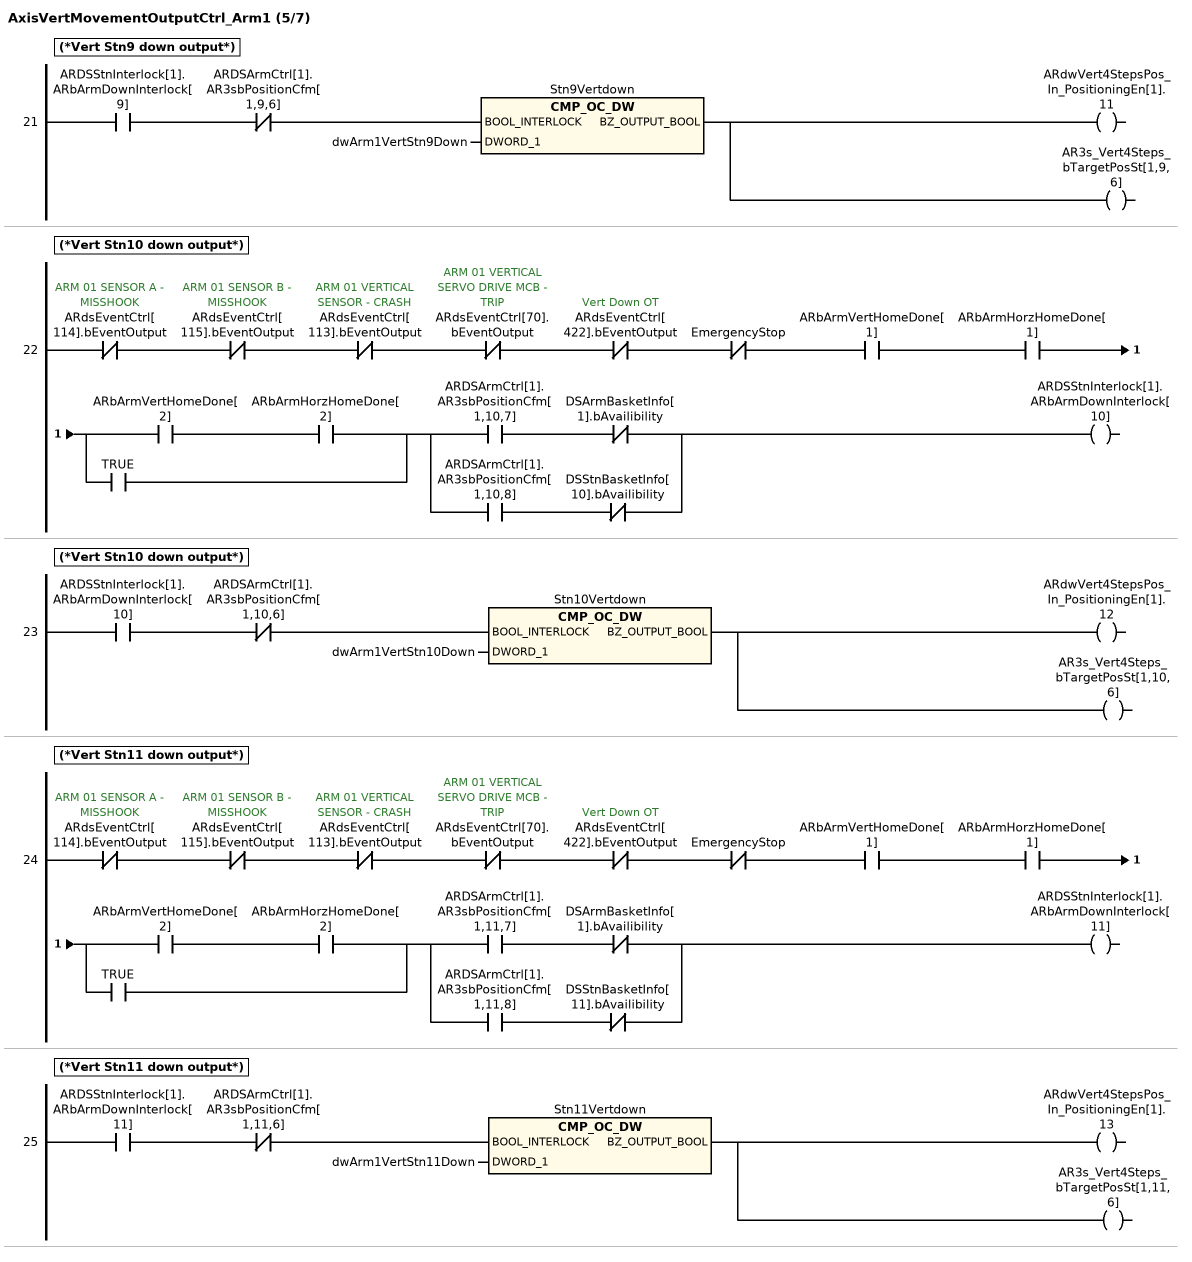
// NETWORK 21
// label: (*Vert Stn9 down output*)
Stn9Vertdown(BOOL_INTERLOCK := ARDSStnInterlock[1].ARbArmDownInterlock[9] AND NOT ARDSArmCtrl[1].AR3sbPositionCfm[1,9,6], DWORD_1 := dwArm1VertStn9Down); // CMP_OC_DW
ARdwVert4StepsPos_In_PositioningEn[1].11 := Stn9Vertdown.BZ_OUTPUT_BOOL;
AR3s_Vert4Steps_bTargetPosSt[1,9,6] := Stn9Vertdown.BZ_OUTPUT_BOOL;

// NETWORK 22
//   ARdsEventCtrl[114].bEventOutput: ARM 01 SENSOR A - MISSHOOK
//   ARdsEventCtrl[115].bEventOutput: ARM 01 SENSOR B - MISSHOOK
//   ARdsEventCtrl[113].bEventOutput: ARM 01 VERTICAL SENSOR - CRASH
//   ARdsEventCtrl[70].bEventOutput: ARM 01 VERTICAL SERVO DRIVE MCB - TRIP
//   ARdsEventCtrl[422].bEventOutput: Vert Down OT
// label: (*Vert Stn10 down output*)
ARDSStnInterlock[1].ARbArmDownInterlock[10] := (NOT ARdsEventCtrl[114].bEventOutput AND NOT ARdsEventCtrl[115].bEventOutput AND NOT ARdsEventCtrl[113].bEventOutput AND NOT ARdsEventCtrl[70].bEventOutput AND NOT ARdsEventCtrl[422].bEventOutput AND NOT EmergencyStop) AND ARbArmVertHomeDone[1] AND ARbArmHorzHomeDone[1] AND (ARbArmVertHomeDone[2] AND ARbArmHorzHomeDone[2] OR TRUE) AND (ARDSArmCtrl[1].AR3sbPositionCfm[1,10,7] AND NOT DSArmBasketInfo[1].bAvailibility OR ARDSArmCtrl[1].AR3sbPositionCfm[1,10,8] AND NOT DSStnBasketInfo[10].bAvailibility);

// NETWORK 23
// label: (*Vert Stn10 down output*)
Stn10Vertdown(BOOL_INTERLOCK := ARDSStnInterlock[1].ARbArmDownInterlock[10] AND NOT ARDSArmCtrl[1].AR3sbPositionCfm[1,10,6], DWORD_1 := dwArm1VertStn10Down); // CMP_OC_DW
ARdwVert4StepsPos_In_PositioningEn[1].12 := Stn10Vertdown.BZ_OUTPUT_BOOL;
AR3s_Vert4Steps_bTargetPosSt[1,10,6] := Stn10Vertdown.BZ_OUTPUT_BOOL;

// NETWORK 24
//   ARdsEventCtrl[114].bEventOutput: ARM 01 SENSOR A - MISSHOOK
//   ARdsEventCtrl[115].bEventOutput: ARM 01 SENSOR B - MISSHOOK
//   ARdsEventCtrl[113].bEventOutput: ARM 01 VERTICAL SENSOR - CRASH
//   ARdsEventCtrl[70].bEventOutput: ARM 01 VERTICAL SERVO DRIVE MCB - TRIP
//   ARdsEventCtrl[422].bEventOutput: Vert Down OT
// label: (*Vert Stn11 down output*)
ARDSStnInterlock[1].ARbArmDownInterlock[11] := (NOT ARdsEventCtrl[114].bEventOutput AND NOT ARdsEventCtrl[115].bEventOutput AND NOT ARdsEventCtrl[113].bEventOutput AND NOT ARdsEventCtrl[70].bEventOutput AND NOT ARdsEventCtrl[422].bEventOutput AND NOT EmergencyStop) AND ARbArmVertHomeDone[1] AND ARbArmHorzHomeDone[1] AND (ARbArmVertHomeDone[2] AND ARbArmHorzHomeDone[2] OR TRUE) AND (ARDSArmCtrl[1].AR3sbPositionCfm[1,11,7] AND NOT DSArmBasketInfo[1].bAvailibility OR ARDSArmCtrl[1].AR3sbPositionCfm[1,11,8] AND NOT DSStnBasketInfo[11].bAvailibility);

// NETWORK 25
// label: (*Vert Stn11 down output*)
Stn11Vertdown(BOOL_INTERLOCK := ARDSStnInterlock[1].ARbArmDownInterlock[11] AND NOT ARDSArmCtrl[1].AR3sbPositionCfm[1,11,6], DWORD_1 := dwArm1VertStn11Down); // CMP_OC_DW
ARdwVert4StepsPos_In_PositioningEn[1].13 := Stn11Vertdown.BZ_OUTPUT_BOOL;
AR3s_Vert4Steps_bTargetPosSt[1,11,6] := Stn11Vertdown.BZ_OUTPUT_BOOL;

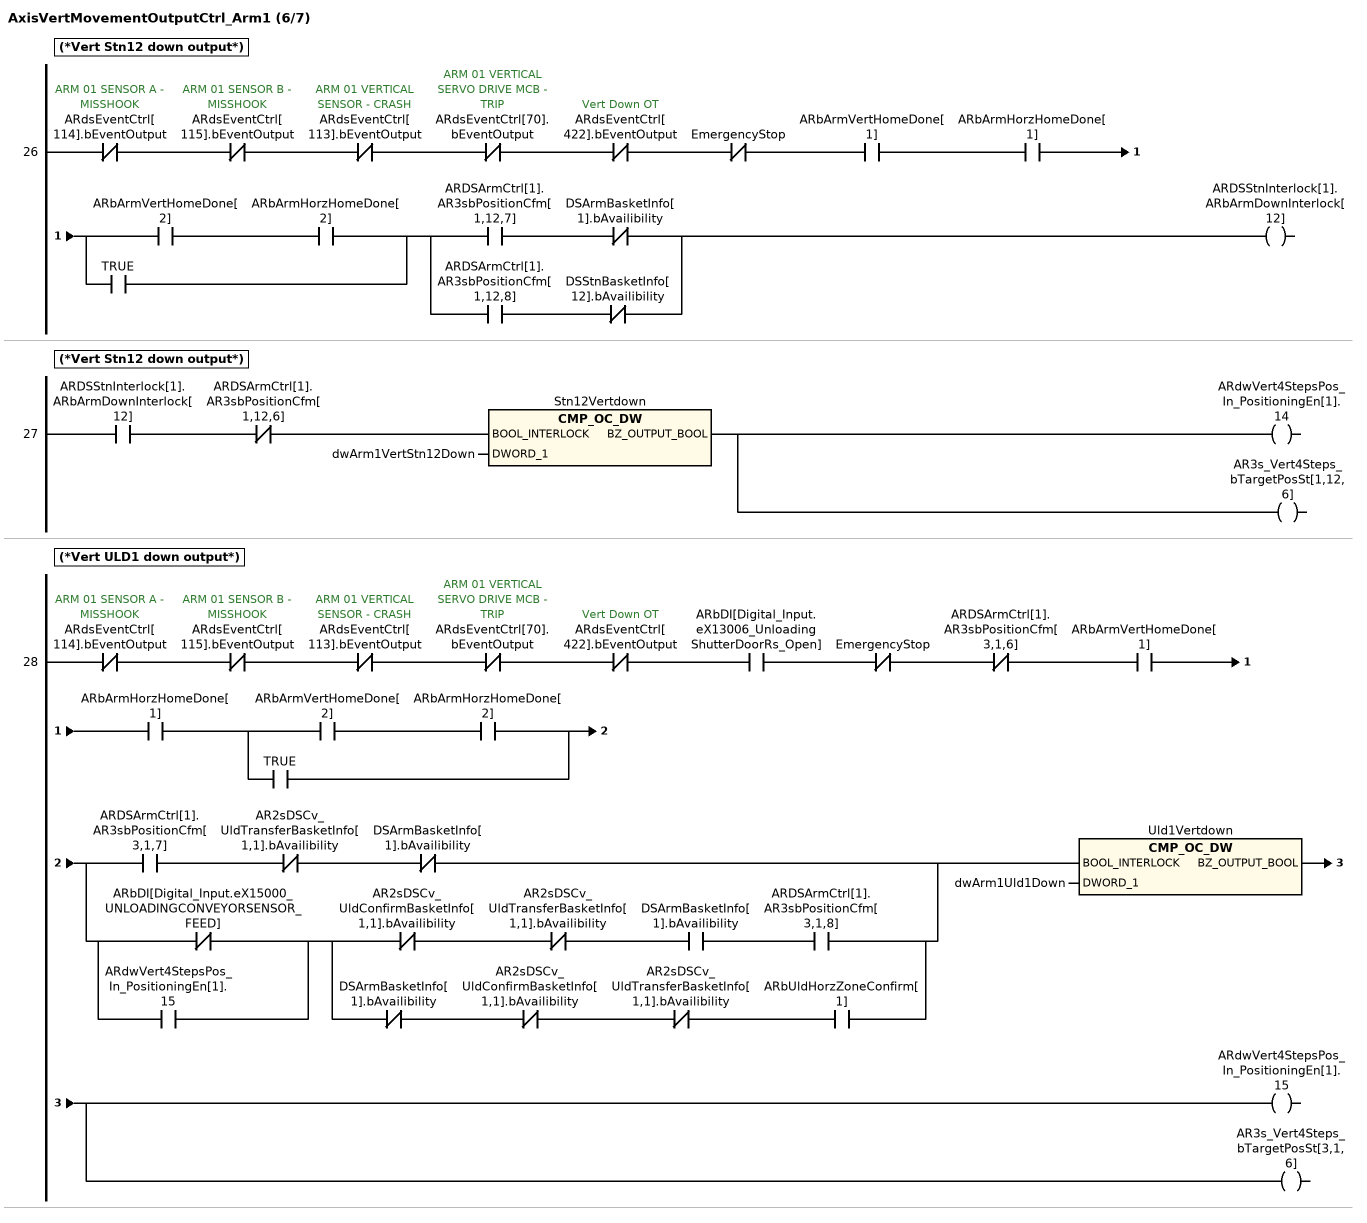
// NETWORK 26
//   ARdsEventCtrl[114].bEventOutput: ARM 01 SENSOR A - MISSHOOK
//   ARdsEventCtrl[115].bEventOutput: ARM 01 SENSOR B - MISSHOOK
//   ARdsEventCtrl[113].bEventOutput: ARM 01 VERTICAL SENSOR - CRASH
//   ARdsEventCtrl[70].bEventOutput: ARM 01 VERTICAL SERVO DRIVE MCB - TRIP
//   ARdsEventCtrl[422].bEventOutput: Vert Down OT
// label: (*Vert Stn12 down output*)
ARDSStnInterlock[1].ARbArmDownInterlock[12] := (NOT ARdsEventCtrl[114].bEventOutput AND NOT ARdsEventCtrl[115].bEventOutput AND NOT ARdsEventCtrl[113].bEventOutput AND NOT ARdsEventCtrl[70].bEventOutput AND NOT ARdsEventCtrl[422].bEventOutput AND NOT EmergencyStop) AND ARbArmVertHomeDone[1] AND ARbArmHorzHomeDone[1] AND (ARbArmVertHomeDone[2] AND ARbArmHorzHomeDone[2] OR TRUE) AND (ARDSArmCtrl[1].AR3sbPositionCfm[1,12,7] AND NOT DSArmBasketInfo[1].bAvailibility OR ARDSArmCtrl[1].AR3sbPositionCfm[1,12,8] AND NOT DSStnBasketInfo[12].bAvailibility);

// NETWORK 27
// label: (*Vert Stn12 down output*)
Stn12Vertdown(BOOL_INTERLOCK := ARDSStnInterlock[1].ARbArmDownInterlock[12] AND NOT ARDSArmCtrl[1].AR3sbPositionCfm[1,12,6], DWORD_1 := dwArm1VertStn12Down); // CMP_OC_DW
ARdwVert4StepsPos_In_PositioningEn[1].14 := Stn12Vertdown.BZ_OUTPUT_BOOL;
AR3s_Vert4Steps_bTargetPosSt[1,12,6] := Stn12Vertdown.BZ_OUTPUT_BOOL;

// NETWORK 28
//   ARdsEventCtrl[114].bEventOutput: ARM 01 SENSOR A - MISSHOOK
//   ARdsEventCtrl[115].bEventOutput: ARM 01 SENSOR B - MISSHOOK
//   ARdsEventCtrl[113].bEventOutput: ARM 01 VERTICAL SENSOR - CRASH
//   ARdsEventCtrl[70].bEventOutput: ARM 01 VERTICAL SERVO DRIVE MCB - TRIP
//   ARdsEventCtrl[422].bEventOutput: Vert Down OT
// label: (*Vert ULD1 down output*)
Uld1Vertdown(BOOL_INTERLOCK := (NOT ARdsEventCtrl[114].bEventOutput AND NOT ARdsEventCtrl[115].bEventOutput AND NOT ARdsEventCtrl[113].bEventOutput AND NOT ARdsEventCtrl[70].bEventOutput AND NOT ARdsEventCtrl[422].bEventOutput AND ARbDI[Digital_Input.eX13006_UnloadingShutterDoorRs_Open] AND NOT EmergencyStop) AND NOT ARDSArmCtrl[1].AR3sbPositionCfm[3,1,6] AND ARbArmVertHomeDone[1] AND ARbArmHorzHomeDone[1] AND (ARbArmVertHomeDone[2] AND ARbArmHorzHomeDone[2] OR TRUE) AND (ARDSArmCtrl[1].AR3sbPositionCfm[3,1,7] AND NOT AR2sDSCv_UldTransferBasketInfo[1,1].bAvailibility AND NOT DSArmBasketInfo[1].bAvailibility OR (NOT ARbDI[Digital_Input.eX15000_UNLOADINGCONVEYORSENSOR_FEED] OR ARdwVert4StepsPos_In_PositioningEn[1].15) AND (NOT AR2sDSCv_UldConfirmBasketInfo[1,1].bAvailibility AND NOT AR2sDSCv_UldTransferBasketInfo[1,1].bAvailibility AND DSArmBasketInfo[1].bAvailibility AND ARDSArmCtrl[1].AR3sbPositionCfm[3,1,8] OR NOT DSArmBasketInfo[1].bAvailibility AND NOT AR2sDSCv_UldConfirmBasketInfo[1,1].bAvailibility AND NOT AR2sDSCv_UldTransferBasketInfo[1,1].bAvailibility AND ARbUldHorzZoneConfirm[1])), DWORD_1 := dwArm1Uld1Down); // CMP_OC_DW
ARdwVert4StepsPos_In_PositioningEn[1].15 := Uld1Vertdown.BZ_OUTPUT_BOOL;
AR3s_Vert4Steps_bTargetPosSt[3,1,6] := Uld1Vertdown.BZ_OUTPUT_BOOL;

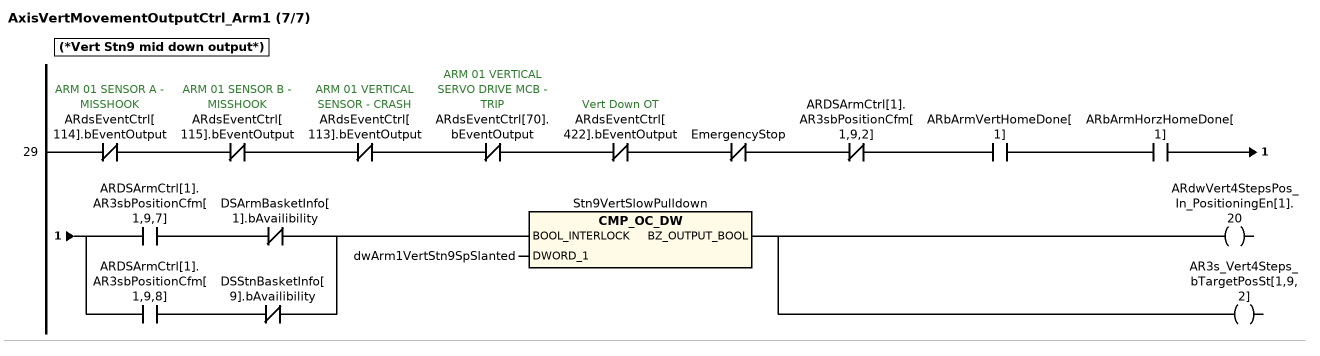
// NETWORK 29
//   ARdsEventCtrl[114].bEventOutput: ARM 01 SENSOR A - MISSHOOK
//   ARdsEventCtrl[115].bEventOutput: ARM 01 SENSOR B - MISSHOOK
//   ARdsEventCtrl[113].bEventOutput: ARM 01 VERTICAL SENSOR - CRASH
//   ARdsEventCtrl[70].bEventOutput: ARM 01 VERTICAL SERVO DRIVE MCB - TRIP
//   ARdsEventCtrl[422].bEventOutput: Vert Down OT
// label: (*Vert Stn9 mid down output*)
Stn9VertSlowPulldown(BOOL_INTERLOCK := (NOT ARdsEventCtrl[114].bEventOutput AND NOT ARdsEventCtrl[115].bEventOutput AND NOT ARdsEventCtrl[113].bEventOutput AND NOT ARdsEventCtrl[70].bEventOutput AND NOT ARdsEventCtrl[422].bEventOutput AND NOT EmergencyStop) AND NOT ARDSArmCtrl[1].AR3sbPositionCfm[1,9,2] AND ARbArmVertHomeDone[1] AND ARbArmHorzHomeDone[1] AND (ARDSArmCtrl[1].AR3sbPositionCfm[1,9,7] AND NOT DSArmBasketInfo[1].bAvailibility OR ARDSArmCtrl[1].AR3sbPositionCfm[1,9,8] AND NOT DSStnBasketInfo[9].bAvailibility), DWORD_1 := dwArm1VertStn9SpSlanted); // CMP_OC_DW
ARdwVert4StepsPos_In_PositioningEn[1].20 := Stn9VertSlowPulldown.BZ_OUTPUT_BOOL;
AR3s_Vert4Steps_bTargetPosSt[1,9,2] := Stn9VertSlowPulldown.BZ_OUTPUT_BOOL;

END_PROGRAM

// ---- POUs/MainProgram/AutoArmCtrl/PnpCtrl_Arm1.TcPOU
PROGRAM PnpCtrl_Arm1

VAR
	fbArmPnpCtrl_Arm1		: fbV2_ArmPnpCtrl;

	fbArmPnpCtrl_Arm1a		: fbV2_1_ArmPnpCtrl;

	Arm1Agi: fbArmSpecialFunctionStore;

	fbVertAgiMovement: fbAxisAgiMovement;

END_VAR

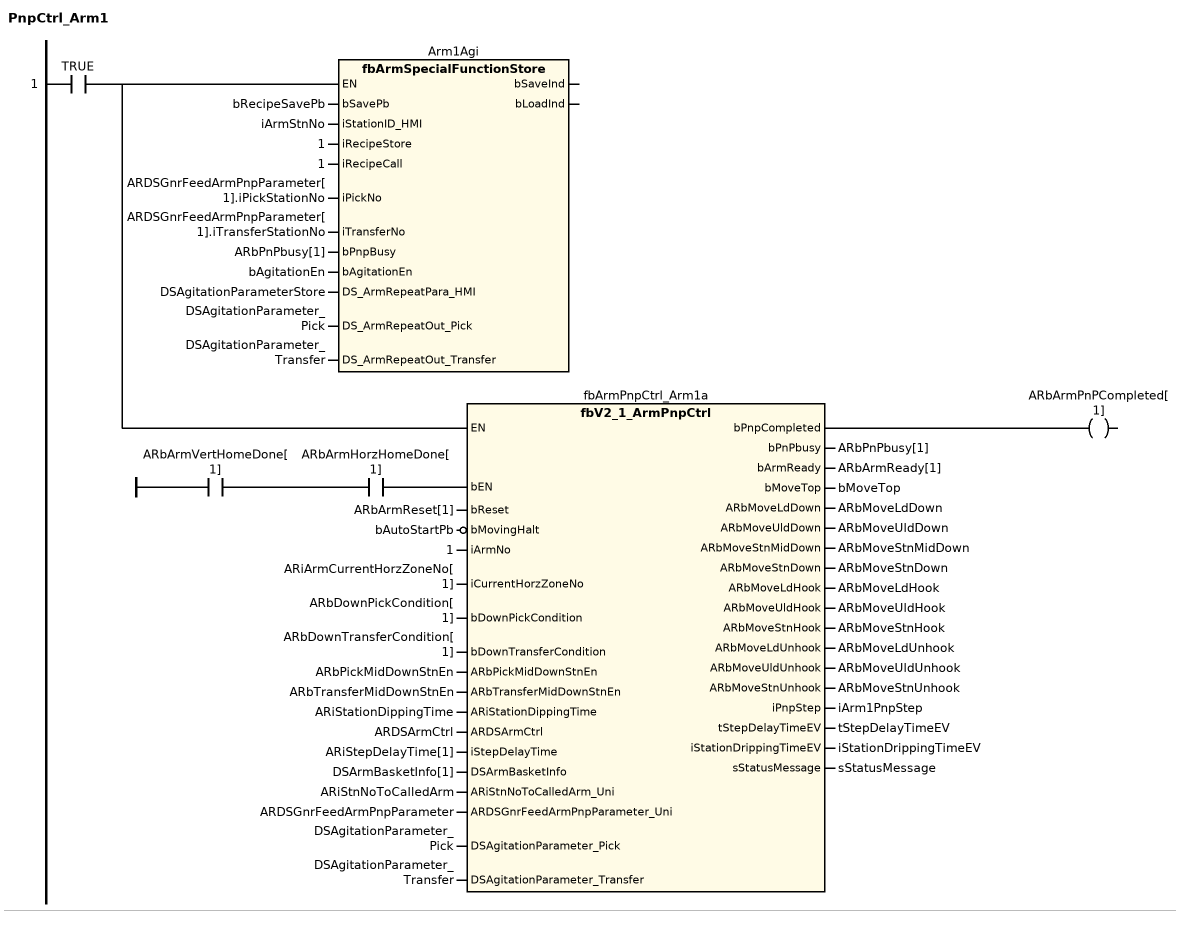
// NETWORK 1
Arm1Agi(
    bSavePb := bRecipeSavePb,
    iStationID_HMI := iArmStnNo,
    iRecipeStore := 1,
    iRecipeCall := 1,
    iPickNo := ARDSGnrFeedArmPnpParameter[1].iPickStationNo,
    iTransferNo := ARDSGnrFeedArmPnpParameter[1].iTransferStationNo,
    bPnpBusy := ARbPnPbusy[1],
    bAgitationEn := bAgitationEn,
    DS_ArmRepeatPara_HMI := DSAgitationParameterStore,
    DS_ArmRepeatOut_Pick := DSAgitationParameter_Pick,
    DS_ArmRepeatOut_Transfer := DSAgitationParameter_Transfer); // fbArmSpecialFunctionStore
fbArmPnpCtrl_Arm1a(
    bEN := ARbArmVertHomeDone[1] AND ARbArmHorzHomeDone[1],
    bReset := ARbArmReset[1],
    bMovingHalt := NOT bAutoStartPb,
    iArmNo := 1,
    iCurrentHorzZoneNo := ARiArmCurrentHorzZoneNo[1],
    bDownPickCondition := ARbDownPickCondition[1],
    bDownTransferCondition := ARbDownTransferCondition[1],
    ARbPickMidDownStnEn := ARbPickMidDownStnEn,
    ARbTransferMidDownStnEn := ARbTransferMidDownStnEn,
    ARiStationDippingTime := ARiStationDippingTime,
    ARDSArmCtrl := ARDSArmCtrl,
    iStepDelayTime := ARiStepDelayTime[1],
    DSArmBasketInfo := DSArmBasketInfo[1],
    ARiStnNoToCalledArm_Uni := ARiStnNoToCalledArm,
    ARDSGnrFeedArmPnpParameter_Uni := ARDSGnrFeedArmPnpParameter,
    DSAgitationParameter_Pick := DSAgitationParameter_Pick,
    DSAgitationParameter_Transfer := DSAgitationParameter_Transfer,
    bPnPbusy => ARbPnPbusy[1],
    bArmReady => ARbArmReady[1],
    bMoveTop => bMoveTop,
    ARbMoveLdDown => ARbMoveLdDown,
    ARbMoveUldDown => ARbMoveUldDown,
    ARbMoveStnMidDown => ARbMoveStnMidDown,
    ARbMoveStnDown => ARbMoveStnDown,
    ARbMoveLdHook => ARbMoveLdHook,
    ARbMoveUldHook => ARbMoveUldHook,
    ARbMoveStnHook => ARbMoveStnHook,
    ARbMoveLdUnhook => ARbMoveLdUnhook,
    ARbMoveUldUnhook => ARbMoveUldUnhook,
    ARbMoveStnUnhook => ARbMoveStnUnhook,
    iPnpStep => iArm1PnpStep,
    tStepDelayTimeEV => tStepDelayTimeEV,
    iStationDrippingTimeEV => iStationDrippingTimeEV,
    sStatusMessage => sStatusMessage); // fbV2_1_ArmPnpCtrl
ARbArmPnPCompleted[1] := fbArmPnpCtrl_Arm1a.bPnpCompleted;

END_PROGRAM

// ---- FBs/B_JKS_NewFB_V2/FBP-ArmCtrlFolder/fbV2_ArmPnpCtrl.TcPOU
FUNCTION_BLOCK fbV2_ArmPnpCtrl

(*************************************************************** Ver.B1 - fbV2_ArmPnpCtrl - 160704 **************************************************************]

 	- at iDSArmZoneStage1 and Stage2, not able to find Ld or Uld Zone due to no forloop and it only rely on ARDSGnrFeedArmPnpParameter. SOLVED																	



[****************************************************************************************************************************************************************************************************)

(*160530 - Change the method of Array Arm Pos Confirm*)


VAR_INPUT
	bEN									:	BOOL;
(*	bExternalCtrl							: 	BOOL;
	bPnPStart							:	BOOL;
	iPickStnNo							:	INT;
	iTransferStnNo						:	INT;
*)	bReset								:	BOOL;
	bMovingHalt							:	BOOL;
	iArmNo								:	INT;
	iCurrentHorzZoneNo					:	INT;
	bDownPickCondition					:	BOOL;
	bDownTransferCondition				:	BOOL;
	ARbPickMidDownStnEn				:	ARRAY [0..iStnQty] OF BOOL;
	ARbTransferMidDownStnEn			:	ARRAY [0..iStnQty] OF BOOL;
	ARiStationDippingTime				:	ARRAY [0..iStnQty] OF INT;
	ARDSArmCtrl							:	ARRAY [0..iArmQty] OF DSV2_ArmPosition;
	iStepDelayTime						:	INT;
END_VAR
VAR_OUTPUT
	bPnpCompleted						:	BOOL;
	bPnPbusy							:	BOOL;
	bArmReady							:  	BOOL;
	bMoveTop							:	BOOL;
	(**)ARbMoveLdDown						:	ARRAY [0..iLdStnQty] OF BOOL;
	(**)ARbMoveUldDown						:	ARRAY [0..iUldStnQty] OF BOOL;
	ARbMoveStnMidDown					:	ARRAY [0..iStnQty] OF BOOL;
	ARbMoveStnDown					:	ARRAY [0..iStnQty] OF BOOL;
	(**)ARbMoveLdHook						:	ARRAY [0..iLdStnQty] OF BOOL;
	(**)ARbMoveUldHook						:	ARRAY [0..iUldStnQty] OF BOOL;
	ARbMoveStnHook					:	ARRAY [0..iStnQty] OF BOOL;
	(**)ARbMoveLdUnhook						:	ARRAY [0..iLdStnQty] OF BOOL;
	(**)ARbMoveUldUnhook						:	ARRAY [0..iUldStnQty] OF BOOL;
	ARbMoveStnUnhook					:	ARRAY [0..iStnQty] OF BOOL;
	iPnpStep								: INT;
	tStepDelayTimeEV					: TIME;
	iStationDrippingTimeEV				: INT;
	sStatusMessage						: STRING(50);

END_VAR

VAR_IN_OUT PERSISTENT
	DSArmBasketInfo	 						: DSV2_BasketInfo;
	ARiStnNoToCalledArm_Uni					: ARRAY [0..iArmQty] OF INT; 									(*Universal*) (* Output - Link with fbArmPnP, Array based on Arm No, The Int will store which Station that calling the Arm*)
	ARDSGnrFeedArmPnpParameter_Uni		: ARRAY [0..iArmQty] OF DSV2_Gnr_CalledArmPnpParameter; 	(*Universal*) (* Output - Link with fbArmPnP, Array based on Current Station No, Arm should move based on this DataStructure Info*)

END_VAR

VAR
	DSEmptyGnrCalledArmPnpParameter : DSV2_Gnr_CalledArmPnpParameter;
	bPnpStart_Read_RE: R_TRIG;
	bPnpStart_Read_FE: F_TRIG;
	iResetFL: INT;
	tStepDelay: TON;
	bStepDelayEn: BOOL;
	iPickStnNoInt: INT;
	iTransferStnNoInt: INT;
	iCurrentHorzZoneNoint: INT;
	bDownPickConditionHR: BOOL;
	bDownTransferConditionHR: BOOL;
	bStationDrippingTimeST: BOOL;
	tStationDrippingTime: TON;
	iStationDrippingTimeInt: INT;
	bPnpStart_Read : BOOL;
	iPickStnNo_Read: INT;
	iPickStnNo_ReadInt: INT;
	iTransferStnNo_Read: INT;
	iTransferStnNo_ReadInt: INT;
	iPnpStep5RE: R_TRIG;
	iDSArmPickStage1: INT;
	iDSArmPickStage2: INT;
	iDSArmTransferStage1: INT;
	iDSArmTransferStage2: INT;
	iDSArmZoneStage1: INT;
	iDSArmZoneStage2: INT;
	iCurrrentZoneMFL: INT;
	iCurrentZoneMFL: INT;
	bLdFound: BOOL;
	bUldFound: BOOL;
	bStnFound: BOOL;
	tStationDrippingTimeEV				: TIME;

END_VAR

(*Mapping*)

iPickStnNo_Read 			:= ARDSGnrFeedArmPnpParameter_Uni[iArmNo].iPickStationNo;
iTransferStnNo_Read 		:= ARDSGnrFeedArmPnpParameter_Uni[iArmNo].iTransferStationNo;

IF ARiStnNoToCalledArm_Uni[iArmNo] <> 0 THEN
bPnpStart_Read := TRUE;
ELSE
bPnpStart_Read := FALSE;
END_IF





(*R_TRIG*)
bPnpStart_Read_RE(CLK:=bPnpStart_Read , Q=> );

(*F_TRIG*)
bPnpStart_Read_FE(CLK:=bPnpStart_Read , Q=> );

(******Station No Conversion******)
(*Pick StnNoConversion*)
IF iPickStnNo_Read = ARiLdStnID[ARDSGnrFeedArmPnpParameter_Uni[iArmNo].iLdGroupNo] THEN
iDSArmPickStage1 := 2;
iDSArmPickStage2 := ARDSGnrFeedArmPnpParameter_Uni[iArmNo].iLdGroupNo;
ELSIF
iPickStnNo_Read = ARiUldStnID[ARDSGnrFeedArmPnpParameter_Uni[iArmNo].iUldGroupNo] THEN
iDSArmPickStage1 := 3;
iDSArmPickStage2 := ARDSGnrFeedArmPnpParameter_Uni[iArmNo].iUldGroupNo;
ELSIF
iPickStnNo_Read >= 1 AND iPickStnNo_Read <= iStnQty THEN
iDSArmPickStage1 := 1;
iDSArmPickStage2 := iPickStnNo_Read;
ELSE
iDSArmPickStage1 := 0;
iDSArmPickStage2 := 0;
END_IF

(*Transfer StnNoConversion*)

IF iTransferStnNo_Read = ARiLdStnID[ARDSGnrFeedArmPnpParameter_Uni[iArmNo].iLdGroupNo] THEN
iDSArmTransferStage1 := 2;
iDSArmTransferStage2 := ARDSGnrFeedArmPnpParameter_Uni[iArmNo].iLdGroupNo;
ELSIF
iTransferStnNo_Read = ARiUldStnID[ARDSGnrFeedArmPnpParameter_Uni[iArmNo].iUldGroupNo]  THEN
iDSArmTransferStage1 := 3;
iDSArmTransferStage2 := ARDSGnrFeedArmPnpParameter_Uni[iArmNo].iUldGroupNo;
ELSIF
iTransferStnNo_Read >= 1 AND iTransferStnNo_Read <= iStnQty THEN
iDSArmTransferStage1 := 1;
iDSArmTransferStage2 := iTransferStnNo_Read;
ELSE
iDSArmTransferStage1 := 0;
iDSArmTransferStage2 := 0;
END_IF


(*iCurrentHorzZoneNo StnNoConversion*)
bLdFound := FALSE;
bUldFound := FALSE;
bStnFound := FALSE;

iCurrrentZoneMFL := 1;
	FOR iCurrentZoneMFL := 1 TO iLdStnQty DO
		IF iCurrentZoneMFL >= 1 AND iCurrentZoneMFL <= iLdStnQty THEN
			IF iCurrentHorzZoneNo = ARiLdStnID[iCurrentZoneMFL] THEN
				iDSArmZoneStage1 := 2;
				iDSArmZoneStage2 := iCurrentZoneMFL;
				bLdFound := TRUE;
			END_IF
		END_IF
	END_FOR

IF NOT bLdFound THEN

iCurrrentZoneMFL := 1;
	FOR iCurrentZoneMFL := 1 TO iUldStnQty DO
		IF iCurrentZoneMFL >= 1 AND iCurrentZoneMFL <= iUldStnQty THEN
			IF iCurrentHorzZoneNo = ARiUldStnID[iCurrentZoneMFL] THEN
				iDSArmZoneStage1 := 3;
				iDSArmZoneStage2 := iCurrentZoneMFL;
				bUldFound := TRUE;
			END_IF
		END_IF
	END_FOR
END_IF

IF NOT bLdFound AND NOT bUldFound THEN

iCurrrentZoneMFL := 1;
	FOR iCurrentZoneMFL := 1 TO iStnQty DO
		IF iCurrentZoneMFL >= 1 AND iCurrentZoneMFL <= iStnQty THEN
			IF iCurrentHorzZoneNo = iCurrentZoneMFL THEN
				iDSArmZoneStage1 := 1;
				iDSArmZoneStage2 := iCurrentZoneMFL;
				bStnFound := TRUE;
			END_IF
		END_IF
	END_FOR
END_IF

(*

IF iCurrentHorzZoneNo = ARiLdStnID[ARDSGnrFeedArmPnpParameter_Uni[iArmNo].iLdGroupNo] THEN
iDSArmZoneStage1 := 2;
iDSArmZoneStage2 := ARDSGnrFeedArmPnpParameter_Uni[iArmNo].iLdGroupNo;
ELSIF
iCurrentHorzZoneNo = ARiUldStnID[ARDSGnrFeedArmPnpParameter_Uni[iArmNo].iUldGroupNo] THEN
iDSArmZoneStage1 := 3;
iDSArmZoneStage2 := ARDSGnrFeedArmPnpParameter_Uni[iArmNo].iUldGroupNo;
ELSIF
iCurrentHorzZoneNo >= 1 AND iCurrentHorzZoneNo <= iStnQty THEN
iDSArmZoneStage1 := 1;
iDSArmZoneStage2 := iCurrentHorzZoneNo;
ELSE*)
IF NOT bStnFound AND NOT bUldFound AND NOT bLdFound THEN
iDSArmZoneStage1 := 0;
iDSArmZoneStage2 := 0;
END_IF




(******Sequence Start******)
(*PnpStep Rising Edge*)
iPnpStep5RE(CLK:=iPnpStep = 5 , Q=> );
(*Step Delay Timer*)
tStepDelay(IN:=bEN AND bPnpStart_Read AND bStepDelayEn , PT:=INT_TO_TIME(iStepDelayTime*1000) , Q=> , ET=>tStepDelayTimeEV );

(*Station Dripping Timer*)
IF iPickStnNo_Read >= 1 AND iPickStnNo_Read <= iStnQty THEN
iStationDrippingTimeInt := ARiStationDippingTime[iPickStnNo_Read];
ELSE
iStationDrippingTimeInt := 0;
END_IF

tStationDrippingTime(IN:=bEN AND bPnpStart_Read AND bStationDrippingTimeST , PT:=DINT_TO_TIME(INT_TO_DINT(iStationDrippingTimeInt)*1000) , Q=> , ET=>tStationDrippingTimeEV );

IF iPnpStep = 5 AND ( iStationDrippingTimeInt > DINT_TO_INT(TIME_TO_DINT(tStationDrippingTimeEV)/1000) )THEN
iStationDrippingTimeEV :=iStationDrippingTimeInt - DINT_TO_INT(TIME_TO_DINT(tStationDrippingTimeEV)/1000);
ELSE
iStationDrippingTimeEV :=0;
END_IF

(*Waiting Start Signal and Condition*)
IF bEN  AND NOT bReset THEN

		IF bPnpStart_Read_RE.Q AND iPickStnNo_Read > 0 AND iTransferStnNo_Read > 0 THEN
		iPnpStep := 1;
		bPnPbusy := TRUE;
		END_IF


		CASE iPnpStep OF

		10: (*Completed*)
		bPnpCompleted:= TRUE;
		bPnPbusy := FALSE;


		9: (*Move Vertical Top Pos*)

			IF NOT ARDSArmCtrl[iArmNo].AR3sbPositionCfm[iDSArmTransferStage1,iDSArmTransferStage2,1] THEN
			bMoveTop := TRUE;
			ELSE
			bMoveTop := FALSE;
			bStepDelayEn := TRUE;
			END_IF

			IF ARDSArmCtrl[iArmNo].AR3sbPositionCfm[iDSArmTransferStage1,iDSArmTransferStage2,1] AND tStepDelay.Q AND NOT bMovingHalt THEN
			bStepDelayEn := FALSE;
			iPnpStep := 10;
			END_IF

			IF NOT ARDSArmCtrl[iArmNo].AR3sbPositionCfm[iDSArmTransferStage1,iDSArmTransferStage2,7] AND NOT bMovingHalt THEN
			bStepDelayEn := FALSE;
			iPnpStep := 8;
			END_IF


		8: (*At Transfer Station - Unhook*)

			IF NOT ARDSArmCtrl[iArmNo].AR3sbPositionCfm[iDSArmTransferStage1,iDSArmTransferStage2,7] (*AR3sbArmPositionCFM[iArmNo,iTransferStnNo_ReadInt,1]*) THEN

				IF iDSArmTransferStage1 = 2 THEN
				ARbMoveLdUnhook[iDSArmTransferStage2] := TRUE;
				END_IF

				IF iDSArmTransferStage1 = 3 THEN
				ARbMoveUldUnhook[iDSArmTransferStage2] := TRUE;
				END_IF

				IF iDSArmTransferStage1= 1 THEN
				ARbMoveStnUnhook[iDSArmTransferStage2] := TRUE;
				END_IF

			ELSE

				IF iDSArmTransferStage1= 1 THEN
				ARbMoveStnUnhook[iDSArmTransferStage2] := FALSE;
				ELSIF iDSArmTransferStage1= 2 THEN
				ARbMoveLdUnhook[iDSArmTransferStage2] := FALSE;
				ELSIF iDSArmTransferStage1= 3 THEN
				ARbMoveUldUnhook[iDSArmTransferStage2] := FALSE;
				END_IF

				bStepDelayEn := TRUE;

			END_IF

			IF ARDSArmCtrl[iArmNo].AR3sbPositionCfm[iDSArmTransferStage1,iDSArmTransferStage2,7] AND tStepDelay.Q AND NOT bMovingHalt THEN
			bStepDelayEn := FALSE;
			iPnpStep := 9;
			END_IF


			IF
			(*bDownTransferConditionHR AND*) NOT ARbTransferMidDownStnEn[iTransferStnNo_Read] AND NOT ARDSArmCtrl[iArmNo].AR3sbPositionCfm[iDSArmTransferStage1,iDSArmTransferStage2,6]
			OR
			(*bDownTransferConditionHR AND*) ARbTransferMidDownStnEn[iTransferStnNo_Read] AND NOT ARDSArmCtrl[iArmNo].AR3sbPositionCfm[iDSArmTransferStage1,iDSArmTransferStage2,2]
			THEN
				IF iDSArmTransferStage1 = 1 THEN
				ARbMoveStnMidDown[iDSArmTransferStage2] := FALSE;
				ARbMoveStnDown[iDSArmTransferStage2] := FALSE;
				ELSIF iDSArmTransferStage1 = 2 THEN
				ARbMoveLdDown[iDSArmTransferStage2] := FALSE;
				ELSIF iDSArmTransferStage1 = 3 THEN
				ARbMoveUldDown[iDSArmTransferStage2] := FALSE;
				END_IF

				bStepDelayEn := TRUE;

				IF tStepDelay.Q AND NOT bMovingHalt THEN
				bStepDelayEn := FALSE;
				bDownTransferConditionHR := FALSE;
				iPnpStep := 7;
				END_IF

			END_IF

		7: (*Move Vertical Down Pos*)

		IF bDownTransferCondition THEN
		bDownTransferConditionHR := TRUE;
		END_IF

			IF bDownTransferConditionHR AND NOT ARbTransferMidDownStnEn[iTransferStnNo_Read] AND NOT ARDSArmCtrl[iArmNo].AR3sbPositionCfm[iDSArmTransferStage1,iDSArmTransferStage2,6] THEN

				IF iDSArmTransferStage1 = 2 THEN
				ARbMoveLdDown[iDSArmTransferStage2] := TRUE;
				END_IF

				IF iDSArmTransferStage1 = 3 THEN
				ARbMoveUldDown[iDSArmTransferStage2] := TRUE;
				END_IF

				IF iDSArmTransferStage1 = 1  THEN
				ARbMoveStnDown[iDSArmTransferStage2] := TRUE;
				END_IF

			ELSIF bDownTransferConditionHR AND ARbTransferMidDownStnEn[iTransferStnNo_Read] AND NOT ARDSArmCtrl[iArmNo].AR3sbPositionCfm[iDSArmTransferStage1,iDSArmTransferStage2,2] THEN

				IF iDSArmTransferStage1 = 1 THEN
				ARbMoveStnMidDown[iDSArmTransferStage2] := TRUE;
				END_IF

			END_IF

			IF
			(*bDownTransferConditionHR AND*) NOT ARbTransferMidDownStnEn[iTransferStnNo_Read] AND ARDSArmCtrl[iArmNo].AR3sbPositionCfm[iDSArmTransferStage1,iDSArmTransferStage2,6]
			OR
			(*bDownTransferConditionHR AND*) ARbTransferMidDownStnEn[iTransferStnNo_Read] AND ARDSArmCtrl[iArmNo].AR3sbPositionCfm[iDSArmTransferStage1,iDSArmTransferStage2,2]
			THEN
				IF iDSArmTransferStage1 = 1 THEN
				ARbMoveStnMidDown[iDSArmTransferStage2] := FALSE;
				ARbMoveStnDown[iDSArmTransferStage2] := FALSE;
				ELSIF iDSArmTransferStage1 = 2 THEN
				ARbMoveLdDown[iDSArmTransferStage2] := FALSE;
				ELSIF iDSArmTransferStage1 = 3 THEN
				ARbMoveUldDown[iDSArmTransferStage2] := FALSE;
				END_IF

				bStepDelayEn := TRUE;

				IF tStepDelay.Q AND NOT bMovingHalt THEN
				bStepDelayEn := FALSE;
				bDownTransferConditionHR := FALSE;
				iPnpStep := 8;
				END_IF

			END_IF

			IF NOT ARDSArmCtrl[iArmNo].AR3sbPositionCfm[iDSArmTransferStage1,iDSArmTransferStage2,8] AND tStepDelay.Q AND NOT bMovingHalt THEN
			bStepDelayEn := FALSE;
			iPnpStep := 6;
			END_IF


		6: (*Move to Transfer Station - Horizontal Hook Movement*)

			IF NOT ARDSArmCtrl[iArmNo].AR3sbPositionCfm[iDSArmTransferStage1,iDSArmTransferStage2,8] (*AR3sbArmPositionCFM[iArmNo,iTransferStnNo_ReadInt,3]*) THEN

				IF iDSArmTransferStage1 = 2 THEN
				ARbMoveLdHook[iDSArmTransferStage2] := TRUE;
				END_IF

				IF iDSArmTransferStage1 = 3 THEN
				ARbMoveUldHook[iDSArmTransferStage2] := TRUE;
				END_IF

				IF iDSArmTransferStage1 = 1 THEN
				ARbMoveStnHook[iDSArmTransferStage2] := TRUE;
				END_IF

			ELSE

				IF iDSArmTransferStage1 = 1THEN
				ARbMoveStnHook[iDSArmTransferStage2] := FALSE;
				ELSIF iDSArmTransferStage1 = 2 THEN
				ARbMoveLdHook[iDSArmTransferStage2] := FALSE;
				ELSIF iDSArmTransferStage1 = 3 THEN
				ARbMoveUldHook[iDSArmTransferStage2] := FALSE;
				END_IF

				bStepDelayEn := TRUE;

			END_IF

			IF ARDSArmCtrl[iArmNo].AR3sbPositionCfm[iDSArmTransferStage1,iDSArmTransferStage2,8] AND tStepDelay.Q AND NOT bMovingHalt THEN
			bStepDelayEn := FALSE;
			iPnpStep := 7;
			END_IF

			IF NOT ARDSArmCtrl[iArmNo].AR3sbPositionCfm[iDSArmPickStage1,iDSArmPickStage2,1] AND NOT bMovingHalt THEN
			bStepDelayEn := FALSE;
			iPnpStep := 5;
			END_IF


		5: (*Move Vertical Top Pos*)

			(*Addtional Task - Push Station Sequence Recipe No from GnrPnpParameter to Basket Info*)
			DSArmBasketInfo.iStationSeqenceRecipeNo := ARDSGnrFeedArmPnpParameter_Uni[iArmNo].iStnSeqRecipeNo;
			IF iPnpStep5RE.Q THEN
			DSArmBasketInfo.iProductRecipeStepNo := DSArmBasketInfo.iProductRecipeStepNo + 1;
			END_IF


			IF NOT ARDSArmCtrl[iArmNo].AR3sbPositionCfm[iDSArmPickStage1,iDSArmPickStage2,1] THEN
			bMoveTop := TRUE;
			ELSE
			bMoveTop := FALSE;
			bStationDrippingTimeST := TRUE;
			END_IF

			IF bStationDrippingTimeST AND tStationDrippingTime.Q THEN
			bStepDelayEn := TRUE;
			END_IF

			IF ARDSArmCtrl[iArmNo].AR3sbPositionCfm[iDSArmPickStage1,iDSArmPickStage2,1] AND bStationDrippingTimeST AND tStationDrippingTime.Q AND tStepDelay.Q AND NOT bMovingHalt THEN
			bStepDelayEn := FALSE;
			bStationDrippingTimeST := FALSE;
			iPnpStep := 6;
			END_IF

			IF NOT ARDSArmCtrl[iArmNo].AR3sbPositionCfm[iDSArmPickStage1,iDSArmPickStage2,8]  AND NOT bMovingHalt THEN
			bStepDelayEn := FALSE;
			iPnpStep := 4;
			END_IF



		4: (*At Pick Station - Hook*)

			IF NOT ARDSArmCtrl[iArmNo].AR3sbPositionCfm[iDSArmPickStage1,iDSArmPickStage2,8] THEN

				IF iDSArmPickStage1 = 2 THEN
				ARbMoveLdHook[iDSArmPickStage2] := TRUE;
				END_IF

				IF iDSArmPickStage1 = 3 THEN
				ARbMoveUldHook[iDSArmPickStage2]:= TRUE;
				END_IF

				IF iDSArmPickStage1 = 1 THEN
				ARbMoveStnHook[iDSArmPickStage2] := TRUE;
				END_IF

			ELSE

				IF iDSArmPickStage1 = 1 THEN
				ARbMoveStnHook[iDSArmPickStage2] := FALSE;
				ELSIF iDSArmPickStage1 = 2 THEN
				ARbMoveLdHook[iDSArmPickStage2] := FALSE;
				ELSIF iDSArmPickStage1 = 3 THEN
				ARbMoveUldHook[iDSArmPickStage2] := FALSE;
				END_IF

				bStepDelayEn := TRUE;

			END_IF

			IF ARDSArmCtrl[iArmNo].AR3sbPositionCfm[iDSArmPickStage1,iDSArmPickStage2,8] AND tStepDelay.Q AND NOT bMovingHalt THEN
			bStepDelayEn := FALSE;
			iPnpStep := 5;
			END_IF

			IF
			(*bDownPickConditionHR AND*) NOT ARbPickMidDownStnEn[iPickStnNo_Read] AND NOT  ARDSArmCtrl[iArmNo].AR3sbPositionCfm[iDSArmPickStage1,iDSArmPickStage2,6]
			OR
			(*bDownPickConditionHR AND*) ARbPickMidDownStnEn[iPickStnNo_Read] AND NOT ARDSArmCtrl[iArmNo].AR3sbPositionCfm[iDSArmPickStage1,iDSArmPickStage2,2]
			THEN
				IF iDSArmPickStage1 = 1 THEN
				ARbMoveStnMidDown[iDSArmPickStage2] := FALSE;
				ARbMoveStnDown[iDSArmPickStage2] := FALSE;
				ELSIF iDSArmPickStage1 = 2 THEN
				ARbMoveLdDown[iDSArmPickStage2] := FALSE;
				ELSIF iDSArmPickStage1 = 3 THEN
				ARbMoveUldDown[iDSArmPickStage2] := FALSE;
				END_IF

				bStepDelayEn := TRUE;

				IF tStepDelay.Q AND NOT bMovingHalt THEN
				bStepDelayEn := FALSE;
				bDownPickConditionHR := FALSE;
				iPnpStep := 3;
				END_IF

			END_IF


		3: (*Move Vertical Down Pos*)

		IF bDownPickCondition THEN
		bDownPickConditionHR := TRUE;
		END_IF

			IF bDownPickConditionHR AND NOT ARbPickMidDownStnEn[iPickStnNo_Read] AND NOT ARDSArmCtrl[iArmNo].AR3sbPositionCfm[iDSArmPickStage1,iDSArmPickStage2,6](*AR3sbArmPositionCFM[iArmNo,iPickStnNo_ReadInt,2]*) THEN

				IF iDSArmPickStage1 = 2 THEN
				ARbMoveLdDown[iDSArmPickStage2] := TRUE;
				END_IF

				IF iDSArmPickStage1 = 3 THEN
				ARbMoveUldDown[iDSArmPickStage2] := TRUE;
				END_IF

				IF iDSArmPickStage1 = 1 THEN
				ARbMoveStnDown[iDSArmPickStage2] := TRUE;
				END_IF

			ELSIF bDownPickConditionHR AND ARbPickMidDownStnEn[iPickStnNo_Read] AND NOT ARDSArmCtrl[iArmNo].AR3sbPositionCfm[iDSArmPickStage1,iDSArmPickStage2,2] THEN

				IF iDSArmPickStage1 = 1 THEN
				ARbMoveStnMidDown[iDSArmPickStage2] := TRUE;
				END_IF

			END_IF

			IF
			(*bDownPickConditionHR AND*) NOT ARbPickMidDownStnEn[iPickStnNo_Read] AND ARDSArmCtrl[iArmNo].AR3sbPositionCfm[iDSArmPickStage1,iDSArmPickStage2,6]
			OR
			(*bDownPickConditionHR AND*) ARbPickMidDownStnEn[iPickStnNo_Read] AND ARDSArmCtrl[iArmNo].AR3sbPositionCfm[iDSArmPickStage1,iDSArmPickStage2,2]
			THEN
				IF iDSArmPickStage1 = 1 THEN
				ARbMoveStnMidDown[iDSArmPickStage2] := FALSE;
				ARbMoveStnDown[iDSArmPickStage2] := FALSE;
				ELSIF iDSArmPickStage1 = 2 THEN
				ARbMoveLdDown[iDSArmPickStage2] := FALSE;
				ELSIF iDSArmPickStage1 = 3 THEN
				ARbMoveUldDown[iDSArmPickStage2] := FALSE;
				END_IF

				bStepDelayEn := TRUE;

				IF tStepDelay.Q AND NOT bMovingHalt THEN
				bStepDelayEn := FALSE;
				bDownPickConditionHR := FALSE;
				iPnpStep := 4;
				END_IF

			END_IF

			IF NOT ARDSArmCtrl[iArmNo].AR3sbPositionCfm[iDSArmPickStage1,iDSArmPickStage2,7]  AND NOT bMovingHalt THEN
			bStepDelayEn := FALSE;
			iPnpStep := 2;
			END_IF




		2: (*Move to Pick Station - Horizontal Unhook Movement*)

			IF NOT ARDSArmCtrl[iArmNo].AR3sbPositionCfm[iDSArmPickStage1,iDSArmPickStage2,7] THEN

				IF iDSArmPickStage1 = 2(*ARiLdStnID*) THEN
				ARbMoveLdUnhook[iDSArmPickStage2] := TRUE;
				END_IF

				IF iDSArmPickStage1 = 3(*ARiUldStnID*) THEN
				ARbMoveUldUnhook[iDSArmPickStage2] := TRUE;
				END_IF

				IF iDSArmPickStage1 = 1 (*iPickStnNo_Read >= 1 AND  iPickStnNo_Read <= iStnQty*) THEN
				ARbMoveStnUnhook[iDSArmPickStage2] := TRUE;
				END_IF

			ELSE

				IF iDSArmPickStage1 = 1(*iPickStnNo_Read >= 1 AND  iPickStnNo_Read <= iStnQty*) THEN
				ARbMoveStnUnhook[iDSArmPickStage2] := FALSE;
				ELSIF iDSArmPickStage1 = 2 THEN
				ARbMoveLdUnhook[iDSArmPickStage2] := FALSE;
				ELSIF iDSArmPickStage1 = 3 THEN
				ARbMoveUldUnhook[iDSArmPickStage2] := FALSE;
				END_IF

				bStepDelayEn := TRUE;

			END_IF

			IF ARDSArmCtrl[iArmNo].AR3sbPositionCfm[iDSArmPickStage1,iDSArmPickStage2,7] AND tStepDelay.Q AND NOT bMovingHalt THEN
			bStepDelayEn := FALSE;
			iPnpStep := 3;
			END_IF

(*LKT*)		IF NOT ARDSArmCtrl[iArmNo].AR3sbPositionCfm[iDSArmZoneStage1,iDSArmZoneStage2,1] AND NOT bMovingHalt THEN
			bStepDelayEn := FALSE;
			iPnpStep := 1;
			END_IF

		1: (*Confirm Vertical Top Pos*)

			IF NOT ARDSArmCtrl[iArmNo].AR3sbPositionCfm[iDSArmZoneStage1,iDSArmZoneStage2,1] THEN
			bMoveTop := TRUE;
			ELSE
			bMoveTop := FALSE;
			bStepDelayEn := TRUE;
			END_IF

			IF ARDSArmCtrl[iArmNo].AR3sbPositionCfm[iDSArmZoneStage1,iDSArmZoneStage2,1] AND tStepDelay.Q AND NOT bMovingHalt THEN
			bStepDelayEn := FALSE;
			iPnpStep := 2;
			END_IF

		0:;







		END_CASE


END_IF

(*Message Display*)

IF NOT bEN THEN
sStatusMessage := 'Arm Not Ready - Homing Required';
ELSIF NOT bPnpStart_Read THEN
sStatusMessage := 'Standby';
END_IF

IF iPnpStep = 1 THEN
sStatusMessage := 'Pnp In Progress - Step 1 - Vertical Up Position';

ELSIF iPnpStep = 2 THEN
sStatusMessage := 'Pnp In Progress - Step 2 - Horizontal Move - Pick Unhook Position';

ELSIF iPnpStep = 3 AND NOT bDownPickCondition THEN
sStatusMessage := 'Pnp In Progress - Step 3 - Waiting Down Pick Condition';

ELSIF iPnpStep = 3 AND bDownPickCondition THEN
sStatusMessage := 'Pnp In Progress - Step 3 - Pick Station Vertical Down Position';

ELSIF iPnpStep = 4 THEN
sStatusMessage := 'Pnp In Progress - Step 4 - Horizontal Move - Pick Hook Position';

ELSIF iPnpStep = 5 AND NOT bStationDrippingTimeST THEN
sStatusMessage := 'Pnp In Progress - Step 5 - Pick Station Vertical Up Position';

ELSIF iPnpStep = 5 AND bStationDrippingTimeST THEN
sStatusMessage := 'Pnp In Progress - Step 5 - Dripping Time Counting';

ELSIF iPnpStep = 6 THEN
sStatusMessage := 'Pnp In Progress - Step 6 - Horizontal Move - Transfer Hook Position';

ELSIF iPnpStep = 7 AND NOT bDownTransferCondition THEN
sStatusMessage := 'Pnp In Progress - Step 7 - Waiting Down Transfer Condition';

ELSIF iPnpStep = 7 AND bDownTransferCondition THEN
sStatusMessage := 'Pnp In Progress - Step 7 - Transfer Station Vertical Down Position';

ELSIF iPnpStep = 8 THEN
sStatusMessage := 'Pnp In Progress - Step 8 - Horizontal Move - Transfer Unhook Position';

ELSIF iPnpStep = 9 THEN
sStatusMessage := 'Pnp In Progress - Step 9 - Transfer Station Vertical Up Position';

ELSIF iPnpStep = 10 THEN
sStatusMessage := 'Pnp Completed';
END_IF

(*Arm Pnp Completed*)
IF bPnpCompleted THEN
	ARiStnNoToCalledArm_Uni[iArmNo] 					:= 0;
	ARDSGnrFeedArmPnpParameter_Uni[iArmNo] 		:= DSEmptyGnrCalledArmPnpParameter;
END_IF


(*Arm Ready Bit*)
IF bEN AND NOT bPnpBusy AND NOT bPnpStart_Read THEN
bArmReady	:= TRUE;
ELSE
bArmReady 	:= FALSE;
END_IF


(*Reset Output*)
IF NOT bEN OR bReset OR bPnpStart_Read_FE.Q THEN

	bPnpCompleted 									:= FALSE;
	bPnpBusy										:= FALSE;
	bMoveTop										:= FALSE;
	iPnpStep											:= 0;
	bDownPickConditionHR 							:= FALSE;
	bDownTransferConditionHR 						:= FALSE;
	bStepDelayEn 									:= FALSE;
	ARiStnNoToCalledArm_Uni[iArmNo] 					:= 0;
	ARDSGnrFeedArmPnpParameter_Uni[iArmNo] 		:= DSEmptyGnrCalledArmPnpParameter;

	iResetFL := 1;
	FOR iResetFL := 1 TO iStnQty DO
		IF iResetFL >= 1 AND iResetFL <= iStnQty THEN
			ARbMoveStnMidDown[iResetFL]			:=	FALSE;
			ARbMoveStnDown[iResetFL]				:=	FALSE;
			ARbMoveStnHook[iResetFL]				:=	FALSE;
			ARbMoveStnUnhook[iResetFL]				:=	FALSE;
		END_IF
	END_FOR

	iResetFL := 1;
	FOR iResetFL := 1 TO iLdStnQty DO
		IF iResetFL >= 1 AND iResetFL <= iLdStnQty THEN
			ARbMoveLdDown[iResetFL]					:= FALSE;
			ARbMoveLdHook[iResetFL]					:= FALSE;
			ARbMoveLdUnhook[iResetFL]					:= FALSE;
		END_IF
	END_FOR

	iResetFL := 1;
	FOR iResetFL := 1 TO iUldStnQty DO
		IF iResetFL >= 1 AND iResetFL <= iUldStnQty THEN
			ARbMoveUldDown[iResetFL]					:= FALSE;
			ARbMoveUldHook[iResetFL]					:= FALSE;
			ARbMoveUldUnhook[iResetFL]				:= FALSE;
		END_IF
	END_FOR

END_IF

END_FUNCTION_BLOCK

// ---- FBs/B_JKS_NewFB_V2/fbArmCtrlFolder/fbV2_1_ArmPnpCtrl.TcPOU
FUNCTION_BLOCK fbV2_1_ArmPnpCtrl

(*************************************************************** Ver.B1 - fbV2_ArmPnpCtrl - 160704 **************************************************************]

 	- at iDSArmZoneStage1 and Stage2, not able to find Ld or Uld Zone due to no forloop and it only rely on ARDSGnrFeedArmPnpParameter. SOLVED																	



[****************************************************************************************************************************************************************************************************)

(*160530 - Change the method of Array Arm Pos Confirm*)


VAR_INPUT
	bEN									:	BOOL;
(*	bExternalCtrl							: 	BOOL;
	bPnPStart							:	BOOL;
	iPickStnNo							:	INT;
	iTransferStnNo						:	INT;
*)	bReset								:	BOOL;
	bMovingHalt							:	BOOL;
	iArmNo								:	INT;
	iCurrentHorzZoneNo					:	INT;
	bDownPickCondition					:	BOOL;
	bDownTransferCondition				:	BOOL;
	ARbPickMidDownStnEn				:	ARRAY [0..iStnQty] OF BOOL;
	ARbTransferMidDownStnEn			:	ARRAY [0..iStnQty] OF BOOL;
	ARiStationDippingTime				:	ARRAY [0..iStnQty] OF INT;
	ARDSArmCtrl							:	ARRAY [0..iArmQty] OF DSV2_ArmPosition;
	iStepDelayTime						:	INT;
END_VAR
VAR_OUTPUT
	bPnpCompleted						:	BOOL;
	bPnPbusy							:	BOOL;
	bArmReady							:  	BOOL;
	bMoveTop							:	BOOL;
	(**)ARbMoveLdDown						:	ARRAY [0..iLdStnQty] OF BOOL;
	(**)ARbMoveUldDown						:	ARRAY [0..iUldStnQty] OF BOOL;
	ARbMoveStnMidDown					:	ARRAY [0..iStnQty] OF BOOL;
	ARbMoveStnDown					:	ARRAY [0..iStnQty] OF BOOL;
	(**)ARbMoveLdHook						:	ARRAY [0..iLdStnQty] OF BOOL;
	(**)ARbMoveUldHook						:	ARRAY [0..iUldStnQty] OF BOOL;
	ARbMoveStnHook					:	ARRAY [0..iStnQty] OF BOOL;
	(**)ARbMoveLdUnhook						:	ARRAY [0..iLdStnQty] OF BOOL;
	(**)ARbMoveUldUnhook						:	ARRAY [0..iUldStnQty] OF BOOL;
	ARbMoveStnUnhook					:	ARRAY [0..iStnQty] OF BOOL;
	iPnpStep								: INT;
	tStepDelayTimeEV					: TIME;
	iStationDrippingTimeEV				: INT;
	sStatusMessage						: STRING(50);

END_VAR

VAR_IN_OUT PERSISTENT
	DSArmBasketInfo	 						: DSV2_BasketInfo;
	ARiStnNoToCalledArm_Uni					: ARRAY [0..iArmQty] OF INT; 									(*Universal*) (* Output - Link with fbArmPnP, Array based on Arm No, The Int will store which Station that calling the Arm*)
	ARDSGnrFeedArmPnpParameter_Uni		: ARRAY [0..iArmQty] OF DSV2_Gnr_CalledArmPnpParameter; 	(*Universal*) (* Output - Link with fbArmPnP, Array based on Current Station No, Arm should move based on this DataStructure Info*)

	DSAgitationParameter_Pick				: DSPnpAgitationParameter ; (*Cheah Add*)
	DSAgitationParameter_Transfer			: DSPnpAgitationParameter ; (*Cheah Add*)


END_VAR

VAR
	DSEmptyGnrCalledArmPnpParameter : DSV2_Gnr_CalledArmPnpParameter;
	bPnpStart_Read_RE: R_TRIG;
	bPnpStart_Read_FE: F_TRIG;
	iResetFL: INT;
	tStepDelay: TON;
	bStepDelayEn: BOOL;
	iPickStnNoInt: INT;
	iTransferStnNoInt: INT;
	iCurrentHorzZoneNoint: INT;
	bDownPickConditionHR: BOOL;
	bDownTransferConditionHR: BOOL;
	bStationDrippingTimeST: BOOL;
	tStationDrippingTime: TON;
	iStationDrippingTimeInt: INT;
	bPnpStart_Read : BOOL;
	iPickStnNo_Read: INT;
	iPickStnNo_ReadInt: INT;
	iTransferStnNo_Read: INT;
	iTransferStnNo_ReadInt: INT;
	iPnpStep5RE: R_TRIG;
	iDSArmPickStage1: INT;
	iDSArmPickStage2: INT;
	iDSArmTransferStage1: INT;
	iDSArmTransferStage2: INT;
	iDSArmZoneStage1: INT;
	iDSArmZoneStage2: INT;
	iCurrrentZoneMFL: INT;
	iCurrentZoneMFL: INT;
	bLdFound: BOOL;
	bUldFound: BOOL;
	bStnFound: BOOL;
	CounterRS: R_TRIG;
	iAgitationCounter: INT;
	tStationDrippingTimeEV				: TIME;
END_VAR

(*Mapping*)

iPickStnNo_Read 			:= ARDSGnrFeedArmPnpParameter_Uni[iArmNo].iPickStationNo;
iTransferStnNo_Read 		:= ARDSGnrFeedArmPnpParameter_Uni[iArmNo].iTransferStationNo;

IF ARiStnNoToCalledArm_Uni[iArmNo] <> 0 THEN
bPnpStart_Read := TRUE;
ELSE
bPnpStart_Read := FALSE;
END_IF





(*R_TRIG*)
bPnpStart_Read_RE(CLK:=bPnpStart_Read , Q=> );

(*F_TRIG*)
bPnpStart_Read_FE(CLK:=bPnpStart_Read , Q=> );

(******Station No Conversion******)
(*Pick StnNoConversion*)
IF iPickStnNo_Read = ARiLdStnID[ARDSGnrFeedArmPnpParameter_Uni[iArmNo].iLdGroupNo] THEN
iDSArmPickStage1 := 2;
iDSArmPickStage2 := ARDSGnrFeedArmPnpParameter_Uni[iArmNo].iLdGroupNo;
ELSIF
iPickStnNo_Read = ARiUldStnID[ARDSGnrFeedArmPnpParameter_Uni[iArmNo].iUldGroupNo] THEN
iDSArmPickStage1 := 3;
iDSArmPickStage2 := ARDSGnrFeedArmPnpParameter_Uni[iArmNo].iUldGroupNo;
ELSIF
iPickStnNo_Read >= 1 AND iPickStnNo_Read <= iStnQty THEN
iDSArmPickStage1 := 1;
iDSArmPickStage2 := iPickStnNo_Read;
ELSE
iDSArmPickStage1 := 0;
iDSArmPickStage2 := 0;
END_IF

(*Transfer StnNoConversion*)

IF iTransferStnNo_Read = ARiLdStnID[ARDSGnrFeedArmPnpParameter_Uni[iArmNo].iLdGroupNo] THEN
iDSArmTransferStage1 := 2;
iDSArmTransferStage2 := ARDSGnrFeedArmPnpParameter_Uni[iArmNo].iLdGroupNo;
ELSIF
iTransferStnNo_Read = ARiUldStnID[ARDSGnrFeedArmPnpParameter_Uni[iArmNo].iUldGroupNo]  THEN
iDSArmTransferStage1 := 3;
iDSArmTransferStage2 := ARDSGnrFeedArmPnpParameter_Uni[iArmNo].iUldGroupNo;
ELSIF
iTransferStnNo_Read >= 1 AND iTransferStnNo_Read <= iStnQty THEN
iDSArmTransferStage1 := 1;
iDSArmTransferStage2 := iTransferStnNo_Read;
ELSE
iDSArmTransferStage1 := 0;
iDSArmTransferStage2 := 0;
END_IF


(*iCurrentHorzZoneNo StnNoConversion*)
bLdFound := FALSE;
bUldFound := FALSE;
bStnFound := FALSE;

iCurrrentZoneMFL := 1;
	FOR iCurrentZoneMFL := 1 TO iLdStnQty DO
		IF iCurrentZoneMFL >= 1 AND iCurrentZoneMFL <= iLdStnQty THEN
			IF iCurrentHorzZoneNo = ARiLdStnID[iCurrentZoneMFL] THEN
				iDSArmZoneStage1 := 2;
				iDSArmZoneStage2 := iCurrentZoneMFL;
				bLdFound := TRUE;
			END_IF
		END_IF
	END_FOR

IF NOT bLdFound THEN

iCurrrentZoneMFL := 1;
	FOR iCurrentZoneMFL := 1 TO iUldStnQty DO
		IF iCurrentZoneMFL >= 1 AND iCurrentZoneMFL <= iUldStnQty THEN
			IF iCurrentHorzZoneNo = ARiUldStnID[iCurrentZoneMFL] THEN
				iDSArmZoneStage1 := 3;
				iDSArmZoneStage2 := iCurrentZoneMFL;
				bUldFound := TRUE;
			END_IF
		END_IF
	END_FOR
END_IF

IF NOT bLdFound AND NOT bUldFound THEN

iCurrrentZoneMFL := 1;
	FOR iCurrentZoneMFL := 1 TO iStnQty DO
		IF iCurrentZoneMFL >= 1 AND iCurrentZoneMFL <= iStnQty THEN
			IF iCurrentHorzZoneNo = iCurrentZoneMFL THEN
				iDSArmZoneStage1 := 1;
				iDSArmZoneStage2 := iCurrentZoneMFL;
				bStnFound := TRUE;
			END_IF
		END_IF
	END_FOR
END_IF

(*

IF iCurrentHorzZoneNo = ARiLdStnID[ARDSGnrFeedArmPnpParameter_Uni[iArmNo].iLdGroupNo] THEN
iDSArmZoneStage1 := 2;
iDSArmZoneStage2 := ARDSGnrFeedArmPnpParameter_Uni[iArmNo].iLdGroupNo;
ELSIF
iCurrentHorzZoneNo = ARiUldStnID[ARDSGnrFeedArmPnpParameter_Uni[iArmNo].iUldGroupNo] THEN
iDSArmZoneStage1 := 3;
iDSArmZoneStage2 := ARDSGnrFeedArmPnpParameter_Uni[iArmNo].iUldGroupNo;
ELSIF
iCurrentHorzZoneNo >= 1 AND iCurrentHorzZoneNo <= iStnQty THEN
iDSArmZoneStage1 := 1;
iDSArmZoneStage2 := iCurrentHorzZoneNo;
ELSE*)
IF NOT bStnFound AND NOT bUldFound AND NOT bLdFound THEN
iDSArmZoneStage1 := 0;
iDSArmZoneStage2 := 0;
END_IF




(******Sequence Start******)
(*PnpStep Rising Edge*)
iPnpStep5RE(CLK:=iPnpStep = 5 , Q=> );
(*Step Delay Timer*)
tStepDelay(IN:=bEN AND bPnpStart_Read AND bStepDelayEn , PT:=INT_TO_TIME(iStepDelayTime*1000) , Q=> , ET=>tStepDelayTimeEV );

(*Station Dripping Timer*)
IF iPickStnNo_Read >= 1 AND iPickStnNo_Read <= iStnQty THEN
iStationDrippingTimeInt := ARiStationDippingTime[iPickStnNo_Read];
ELSE
iStationDrippingTimeInt := 0;
END_IF

tStationDrippingTime(IN:=bEN AND bPnpStart_Read AND bStationDrippingTimeST , PT:=DINT_TO_TIME(INT_TO_DINT(iStationDrippingTimeInt)*1000) , Q=> , ET=>tStationDrippingTimeEV );

IF iPnpStep = 5 AND ( iStationDrippingTimeInt > DINT_TO_INT(TIME_TO_DINT(tStationDrippingTimeEV)/1000) )THEN
iStationDrippingTimeEV :=iStationDrippingTimeInt - DINT_TO_INT(TIME_TO_DINT(tStationDrippingTimeEV)/1000);
ELSE
iStationDrippingTimeEV :=0;
END_IF

(*Waiting Start Signal and Condition*)
IF bEN  AND NOT bReset THEN

		IF bPnpStart_Read_RE.Q AND iPickStnNo_Read > 0 AND iTransferStnNo_Read > 0 THEN
		iPnpStep := 1;
		bPnPbusy := TRUE;
		END_IF


		CASE iPnpStep OF


(*======================================================================================================*)
		50:
			IF DSAgitationParameter_Pick.bAgitationComplete THEN
				iPnpStep := 5;
			END_IF

		51:
			IF DSAgitationParameter_Transfer.bAgitationComplete THEN
				iPnpStep := 7;
			END_IF

(*======================================================================================================*)


		10: (*Completed*)
		bPnpCompleted:= TRUE;
		bPnPbusy := FALSE;
		DSAgitationParameter_Pick.bAgitationComplete := FALSE;
		DSAgitationParameter_Transfer.bAgitationComplete := FALSE;
		DSAgitationParameter_Pick.bAgitationInProgress := FALSE;
		DSAgitationParameter_Transfer.bAgitationInProgress := FALSE;

		9: (*Move Vertical Top Pos*)

			IF NOT ARDSArmCtrl[iArmNo].AR3sbPositionCfm[iDSArmTransferStage1,iDSArmTransferStage2,1] THEN
			bMoveTop := TRUE;
			ELSE
			bMoveTop := FALSE;
			bStepDelayEn := TRUE;
			END_IF

			IF ARDSArmCtrl[iArmNo].AR3sbPositionCfm[iDSArmTransferStage1,iDSArmTransferStage2,1] AND tStepDelay.Q AND NOT bMovingHalt THEN
			bStepDelayEn := FALSE;
			iPnpStep := 10;
			END_IF


		8: (*At Transfer Station - Unhook*)
		
			IF NOT ARDSArmCtrl[iArmNo].AR3sbPositionCfm[iDSArmTransferStage1,iDSArmTransferStage2,7] (*AR3sbArmPositionCFM[iArmNo,iTransferStnNo_ReadInt,1]*) THEN
		
				IF iDSArmTransferStage1 = 2 THEN
				ARbMoveLdUnhook[iDSArmTransferStage2] := TRUE;
				END_IF

				IF iDSArmTransferStage1 = 3 THEN
				ARbMoveUldUnhook[iDSArmTransferStage2] := TRUE;
				END_IF

				IF iDSArmTransferStage1= 1 THEN
				ARbMoveStnUnhook[iDSArmTransferStage2] := TRUE;
				END_IF
		
			ELSE
		
				IF iDSArmTransferStage1= 1 THEN
				ARbMoveStnUnhook[iDSArmTransferStage2] := FALSE;
				ELSIF iDSArmTransferStage1= 2 THEN
				ARbMoveLdUnhook[iDSArmTransferStage2] := FALSE;
				ELSIF iDSArmTransferStage1= 3 THEN
				ARbMoveUldUnhook[iDSArmTransferStage2] := FALSE;
				END_IF
		
				bStepDelayEn := TRUE;

			END_IF

			IF ARDSArmCtrl[iArmNo].AR3sbPositionCfm[iDSArmTransferStage1,iDSArmTransferStage2,7] AND tStepDelay.Q AND NOT bMovingHalt THEN
			bStepDelayEn := FALSE;
			iPnpStep := 9;
			END_IF
		

		7: (*Move Vertical Down Pos*)

		IF bDownTransferCondition THEN
		bDownTransferConditionHR := TRUE;
		END_IF

			IF bDownTransferConditionHR AND NOT ARbTransferMidDownStnEn[iTransferStnNo_Read] AND NOT ARDSArmCtrl[iArmNo].AR3sbPositionCfm[iDSArmTransferStage1,iDSArmTransferStage2,6] THEN

				IF iDSArmTransferStage1 = 2 THEN
				ARbMoveLdDown[iDSArmTransferStage2] := TRUE;
				END_IF

				IF iDSArmTransferStage1 = 3 THEN
				ARbMoveUldDown[iDSArmTransferStage2] := TRUE;
				END_IF

				IF iDSArmTransferStage1 = 1  THEN
				ARbMoveStnDown[iDSArmTransferStage2] := TRUE;
				END_IF

			ELSIF bDownTransferConditionHR AND ARbTransferMidDownStnEn[iTransferStnNo_Read] AND NOT ARDSArmCtrl[iArmNo].AR3sbPositionCfm[iDSArmTransferStage1,iDSArmTransferStage2,2] THEN

				IF iDSArmTransferStage1 = 1 THEN
				ARbMoveStnMidDown[iDSArmTransferStage2] := TRUE;
				END_IF

			END_IF

			IF
			(*bDownTransferConditionHR AND*) NOT ARbTransferMidDownStnEn[iTransferStnNo_Read] AND ARDSArmCtrl[iArmNo].AR3sbPositionCfm[iDSArmTransferStage1,iDSArmTransferStage2,6]
			OR
			(*bDownTransferConditionHR AND*) ARbTransferMidDownStnEn[iTransferStnNo_Read] AND ARDSArmCtrl[iArmNo].AR3sbPositionCfm[iDSArmTransferStage1,iDSArmTransferStage2,2]
			THEN
				IF iDSArmTransferStage1 = 1 THEN
				ARbMoveStnMidDown[iDSArmTransferStage2] := FALSE;
				ARbMoveStnDown[iDSArmTransferStage2] := FALSE;
				ELSIF iDSArmTransferStage1 = 2 THEN
				ARbMoveLdDown[iDSArmTransferStage2] := FALSE;
				ELSIF iDSArmTransferStage1 = 3 THEN
				ARbMoveUldDown[iDSArmTransferStage2] := FALSE;
				END_IF

				bStepDelayEn := TRUE;

				IF tStepDelay.Q AND NOT bMovingHalt THEN
				bStepDelayEn := FALSE;
				bDownTransferConditionHR := FALSE;
				iPnpStep := 8;
				END_IF

			END_IF

		6: (*Move to Transfer Station - Horizontal Hook Movement*)
		
			IF NOT ARDSArmCtrl[iArmNo].AR3sbPositionCfm[iDSArmTransferStage1,iDSArmTransferStage2,8] (*AR3sbArmPositionCFM[iArmNo,iTransferStnNo_ReadInt,3]*) THEN

				IF iDSArmTransferStage1 = 2 THEN
				ARbMoveLdHook[iDSArmTransferStage2] := TRUE;
				END_IF

				IF iDSArmTransferStage1 = 3 THEN
				ARbMoveUldHook[iDSArmTransferStage2] := TRUE;
				END_IF

				IF iDSArmTransferStage1 = 1 THEN
				ARbMoveStnHook[iDSArmTransferStage2] := TRUE;
				END_IF

			ELSE
		
				IF iDSArmTransferStage1 = 1THEN
				ARbMoveStnHook[iDSArmTransferStage2] := FALSE;
				ELSIF iDSArmTransferStage1 = 2 THEN
				ARbMoveLdHook[iDSArmTransferStage2] := FALSE;
				ELSIF iDSArmTransferStage1 = 3 THEN
				ARbMoveUldHook[iDSArmTransferStage2] := FALSE;
				END_IF

				bStepDelayEn := TRUE;
		
			END_IF

			IF NOT DSAgitationParameter_Transfer.bTransferRepeatStnEnable AND DSAgitationParameter_Transfer.bSearchFinish  AND ARDSArmCtrl[iArmNo].AR3sbPositionCfm[iDSArmTransferStage1,iDSArmTransferStage2,8] AND tStepDelay.Q AND NOT bMovingHalt THEN
			bStepDelayEn := FALSE;
			iPnpStep := 7;
			END_IF
(*======*)
			IF DSAgitationParameter_Transfer.bTransferRepeatStnEnable AND DSAgitationParameter_Transfer.bSearchFinish  AND NOT DSAgitationParameter_Transfer.bAgitationComplete AND ARDSArmCtrl[iArmNo].AR3sbPositionCfm[iDSArmTransferStage1,iDSArmTransferStage2,8] AND tStepDelay.Q AND NOT bMovingHalt  THEN
			bStepDelayEn := FALSE;
			iPnpStep := 51;
			END_IF


		5: (*Move Vertical Top Pos*)

			(*Addtional Task - Push Station Sequence Recipe No from GnrPnpParameter to Basket Info*)
			DSArmBasketInfo.iStationSeqenceRecipeNo := ARDSGnrFeedArmPnpParameter_Uni[iArmNo].iStnSeqRecipeNo;
			IF iPnpStep5RE.Q THEN
			DSArmBasketInfo.iProductRecipeStepNo := DSArmBasketInfo.iProductRecipeStepNo + 1;
			END_IF


			IF NOT ARDSArmCtrl[iArmNo].AR3sbPositionCfm[iDSArmPickStage1,iDSArmPickStage2,1] THEN
			bMoveTop := TRUE;
			ELSE
			bMoveTop := FALSE;
			bStationDrippingTimeST := TRUE;
			END_IF

			IF bStationDrippingTimeST AND tStationDrippingTime.Q THEN
			bStepDelayEn := TRUE;
			END_IF

			IF ARDSArmCtrl[iArmNo].AR3sbPositionCfm[iDSArmPickStage1,iDSArmPickStage2,1] AND bStationDrippingTimeST AND tStationDrippingTime.Q AND tStepDelay.Q AND NOT bMovingHalt THEN
			bStepDelayEn := FALSE;
			bStationDrippingTimeST := FALSE;
			iPnpStep := 6;
			END_IF


		4: (*At Pick Station - Hook*)

		
			IF NOT ARDSArmCtrl[iArmNo].AR3sbPositionCfm[iDSArmPickStage1,iDSArmPickStage2,8] THEN
		
				IF iDSArmPickStage1 = 2 THEN
				ARbMoveLdHook[iDSArmPickStage2] := TRUE;
				END_IF
		
				IF iDSArmPickStage1 = 3 THEN
				ARbMoveUldHook[iDSArmPickStage2]:= TRUE;
				END_IF

				IF iDSArmPickStage1 = 1 THEN
				ARbMoveStnHook[iDSArmPickStage2] := TRUE;
				END_IF

			ELSE
		
				IF iDSArmPickStage1 = 1 THEN
				ARbMoveStnHook[iDSArmPickStage2] := FALSE;
				ELSIF iDSArmPickStage1 = 2 THEN
				ARbMoveLdHook[iDSArmPickStage2] := FALSE;
				ELSIF iDSArmPickStage1 = 3 THEN
				ARbMoveUldHook[iDSArmPickStage2] := FALSE;
				END_IF

				bStepDelayEn := TRUE;

			END_IF

			IF NOT DSAgitationParameter_Pick.bPickRepeatStnEnable AND DSAgitationParameter_Pick.bSearchFinish AND ARDSArmCtrl[iArmNo].AR3sbPositionCfm[iDSArmPickStage1,iDSArmPickStage2,8] AND tStepDelay.Q AND NOT bMovingHalt THEN
			bStepDelayEn := FALSE;
			iPnpStep := 5;
			END_IF
(*======*)
			IF DSAgitationParameter_Pick.bPickRepeatStnEnable AND DSAgitationParameter_Pick.bSearchFinish AND NOT DSAgitationParameter_Pick.bAgitationComplete  AND ARDSArmCtrl[iArmNo].AR3sbPositionCfm[iDSArmPickStage1,iDSArmPickStage2,8] AND tStepDelay.Q AND NOT bMovingHalt  THEN
			bStepDelayEn := FALSE;
			iPnpStep := 50;
			END_IF


		3: (*Move Vertical Down Pos*)

		IF NOT ARDSArmCtrl[iArmNo].AR3sbPositionCfm[iDSArmPickStage1,iDSArmPickStage2,7] THEN
			iPnpStep := 2;
		END_IF

		IF bDownPickCondition THEN
		bDownPickConditionHR := TRUE;
		END_IF

			IF bDownPickConditionHR AND NOT ARbPickMidDownStnEn[iPickStnNo_Read] AND NOT ARDSArmCtrl[iArmNo].AR3sbPositionCfm[iDSArmPickStage1,iDSArmPickStage2,6](*AR3sbArmPositionCFM[iArmNo,iPickStnNo_ReadInt,2]*) THEN

				IF iDSArmPickStage1 = 2 THEN
				ARbMoveLdDown[iDSArmPickStage2] := TRUE;
				END_IF
		
				IF iDSArmPickStage1 = 3 THEN
				ARbMoveUldDown[iDSArmPickStage2] := TRUE;
				END_IF
		
				IF iDSArmPickStage1 = 1 THEN
				ARbMoveStnDown[iDSArmPickStage2] := TRUE;
				END_IF

			ELSIF bDownPickConditionHR AND ARbPickMidDownStnEn[iPickStnNo_Read] AND NOT ARDSArmCtrl[iArmNo].AR3sbPositionCfm[iDSArmPickStage1,iDSArmPickStage2,2] THEN

				IF iDSArmPickStage1 = 1 THEN
				ARbMoveStnMidDown[iDSArmPickStage2] := TRUE;
				END_IF

			END_IF

			IF
			(*bDownPickConditionHR AND*) NOT ARbPickMidDownStnEn[iPickStnNo_Read] AND ARDSArmCtrl[iArmNo].AR3sbPositionCfm[iDSArmPickStage1,iDSArmPickStage2,6]
			OR
			(*bDownPickConditionHR AND*) ARbPickMidDownStnEn[iPickStnNo_Read] AND ARDSArmCtrl[iArmNo].AR3sbPositionCfm[iDSArmPickStage1,iDSArmPickStage2,2]
			THEN
				IF iDSArmPickStage1 = 1 THEN
				ARbMoveStnMidDown[iDSArmPickStage2] := FALSE;
				ARbMoveStnDown[iDSArmPickStage2] := FALSE;
				ELSIF iDSArmPickStage1 = 2 THEN
				ARbMoveLdDown[iDSArmPickStage2] := FALSE;
				ELSIF iDSArmPickStage1 = 3 THEN
				ARbMoveUldDown[iDSArmPickStage2] := FALSE;
				END_IF

				bStepDelayEn := TRUE;

				IF tStepDelay.Q AND NOT bMovingHalt THEN
				bStepDelayEn := FALSE;
				bDownPickConditionHR := FALSE;
				iPnpStep := 4;
				END_IF

			END_IF


		
		
		2: (*Move to Pick Station - Horizontal Unhook Movement*)

			IF NOT ARDSArmCtrl[iArmNo].AR3sbPositionCfm[iDSArmPickStage1,iDSArmPickStage2,7] THEN

				IF iDSArmPickStage1 = 2(*ARiLdStnID*) THEN
				ARbMoveLdUnhook[iDSArmPickStage2] := TRUE;
				END_IF

				IF iDSArmPickStage1 = 3(*ARiUldStnID*) THEN
				ARbMoveUldUnhook[iDSArmPickStage2] := TRUE;
				END_IF
		
				IF iDSArmPickStage1 = 1 (*iPickStnNo_Read >= 1 AND  iPickStnNo_Read <= iStnQty*) THEN
				ARbMoveStnUnhook[iDSArmPickStage2] := TRUE;
				END_IF
		
			ELSE

				IF iDSArmPickStage1 = 1(*iPickStnNo_Read >= 1 AND  iPickStnNo_Read <= iStnQty*) THEN
				ARbMoveStnUnhook[iDSArmPickStage2] := FALSE;
				ELSIF iDSArmPickStage1 = 2 THEN
				ARbMoveLdUnhook[iDSArmPickStage2] := FALSE;
				ELSIF iDSArmPickStage1 = 3 THEN
				ARbMoveUldUnhook[iDSArmPickStage2] := FALSE;
				END_IF

				bStepDelayEn := TRUE;

			END_IF

			IF ARDSArmCtrl[iArmNo].AR3sbPositionCfm[iDSArmPickStage1,iDSArmPickStage2,7] AND tStepDelay.Q AND NOT bMovingHalt THEN
			bStepDelayEn := FALSE;
			iPnpStep := 3;
			END_IF


		1: (*Confirm Vertical Top Pos*)

			iAgitationCounter := 0;


			IF NOT ARDSArmCtrl[iArmNo].AR3sbPositionCfm[iDSArmZoneStage1,iDSArmZoneStage2,1] THEN
			bMoveTop := TRUE;
			ELSE
			bMoveTop := FALSE;
			bStepDelayEn := TRUE;
			END_IF

			IF ARDSArmCtrl[iArmNo].AR3sbPositionCfm[iDSArmZoneStage1,iDSArmZoneStage2,1] AND tStepDelay.Q AND NOT bMovingHalt THEN
			bStepDelayEn := FALSE;
			iPnpStep := 2;
			END_IF

		0:;







		END_CASE


END_IF

(*Message Display*)

IF NOT bEN THEN
sStatusMessage := 'Arm Not Ready - Homing Required';
ELSIF NOT bPnpStart_Read THEN
sStatusMessage := 'Standby';
END_IF

IF iPnpStep = 1 THEN
sStatusMessage := 'Pnp In Progress - Step 1 - Vertical Up Position';

ELSIF iPnpStep = 2 THEN
sStatusMessage := 'Pnp In Progress - Step 2 - Horizontal Move - Pick Unhook Position';

ELSIF iPnpStep = 3 AND NOT bDownPickCondition THEN
sStatusMessage := 'Pnp In Progress - Step 3 - Waiting Down Pick Condition';

ELSIF iPnpStep = 3 AND bDownPickCondition THEN
sStatusMessage := 'Pnp In Progress - Step 3 - Pick Station Vertical Down Position';

ELSIF iPnpStep = 4 THEN
sStatusMessage := 'Pnp In Progress - Step 4 - Horizontal Move - Pick Hook Position';

ELSIF iPnpStep = 5 AND NOT bStationDrippingTimeST THEN
sStatusMessage := 'Pnp In Progress - Step 5 - Pick Station Vertical Up Position';

ELSIF iPnpStep = 5 AND bStationDrippingTimeST THEN
sStatusMessage := 'Pnp In Progress - Step 5 - Dripping Time Counting';

ELSIF iPnpStep = 6 THEN
sStatusMessage := 'Pnp In Progress - Step 6 - Horizontal Move - Transfer Hook Position';

ELSIF iPnpStep = 7 AND NOT bDownTransferCondition THEN
sStatusMessage := 'Pnp In Progress - Step 7 - Waiting Down Transfer Condition';

ELSIF iPnpStep = 7 AND bDownTransferCondition THEN
sStatusMessage := 'Pnp In Progress - Step 7 - Transfer Station Vertical Down Position';

ELSIF iPnpStep = 8 THEN
sStatusMessage := 'Pnp In Progress - Step 8 - Horizontal Move - Transfer Unhook Position';

ELSIF iPnpStep = 9 THEN
sStatusMessage := 'Pnp In Progress - Step 9 - Transfer Station Vertical Up Position';

ELSIF iPnpStep = 50 THEN
sStatusMessage := 'Pnp In Progress - Step 50 - Agitation In Progress';

ELSIF iPnpStep = 10 THEN
sStatusMessage := 'Pnp Completed';
END_IF

(*Arm Pnp Completed*)
IF bPnpCompleted THEN
	ARiStnNoToCalledArm_Uni[iArmNo] 					:= 0;
	ARDSGnrFeedArmPnpParameter_Uni[iArmNo] 		:= DSEmptyGnrCalledArmPnpParameter;
END_IF


(*Arm Ready Bit*)
IF bEN AND NOT bPnpBusy AND NOT bPnpStart_Read THEN
bArmReady	:= TRUE;
ELSE
bArmReady 	:= FALSE;
END_IF


(*Reset Output*)
IF NOT bEN OR bReset OR bPnpStart_Read_FE.Q THEN

	bPnpCompleted 									:= FALSE;
	bPnpBusy										:= FALSE;
	bMoveTop										:= FALSE;
	iPnpStep											:= 0;
	bDownPickConditionHR 							:= FALSE;
	bDownTransferConditionHR 						:= FALSE;
	bStepDelayEn 									:= FALSE;
	ARiStnNoToCalledArm_Uni[iArmNo] 					:= 0;
	ARDSGnrFeedArmPnpParameter_Uni[iArmNo] 		:= DSEmptyGnrCalledArmPnpParameter;

	iResetFL := 1;
	FOR iResetFL := 1 TO iStnQty DO
		IF iResetFL >= 1 AND iResetFL <= iStnQty THEN
			ARbMoveStnMidDown[iResetFL]			:=	FALSE;
			ARbMoveStnDown[iResetFL]				:=	FALSE;
			ARbMoveStnHook[iResetFL]				:=	FALSE;
			ARbMoveStnUnhook[iResetFL]				:=	FALSE;
		END_IF
	END_FOR

	iResetFL := 1;
	FOR iResetFL := 1 TO iLdStnQty DO
		IF iResetFL >= 1 AND iResetFL <= iLdStnQty THEN
			ARbMoveLdDown[iResetFL]					:= FALSE;
			ARbMoveLdHook[iResetFL]					:= FALSE;
			ARbMoveLdUnhook[iResetFL]					:= FALSE;
		END_IF
	END_FOR

	iResetFL := 1;
	FOR iResetFL := 1 TO iUldStnQty DO
		IF iResetFL >= 1 AND iResetFL <= iUldStnQty THEN
			ARbMoveUldDown[iResetFL]					:= FALSE;
			ARbMoveUldHook[iResetFL]					:= FALSE;
			ARbMoveUldUnhook[iResetFL]				:= FALSE;
		END_IF
	END_FOR

END_IF

END_FUNCTION_BLOCK

// ---- FBs/FB_Others TBD/fbArmSpecialFunctionStore.TcPOU
FUNCTION_BLOCK fbArmSpecialFunctionStore
VAR_INPUT

	bSavePb			: BOOL;
	iStationID_HMI		: INT;
	iRecipeStore			: INT;
	iRecipeCall			: INT;
	iPickNo				: INT;
	iTransferNo			: INT;
	bPnpBusy			: BOOL;
	bAgitationEn			: BOOL;

END_VAR
VAR_OUTPUT
	bSaveInd			: BOOL;
	bLoadInd			: BOOL;

END_VAR
VAR_IN_OUT

	DS_ArmRepeatPara_HMI			: DSPnpAgitationParameter;
	DS_ArmRepeatOut_Pick		: DSPnpAgitationParameter;
	DS_ArmRepeatOut_Transfer	: DSPnpAgitationParameter;
END_VAR

VAR
	R_TRIG1: R_TRIG;
	iStep: INT;
	iFL1: INT;
	R_TRIG2: R_TRIG;
	R_TRIG3: R_TRIG;

	TON50: TON;
	iBufferRecipe: INT;

	DSArArmRepeatParaEmpty : ARRAY [1..iProductRecipeArrayQty, 1..iStnQty] OF DSPnpAgitationParameter;
	DS_ArmRepeatOut_Empty		: DSPnpAgitationParameter;

	iBufferStnID: INT;
END_VAR

VAR PERSISTENT

	DSArArmRepeatParaStore : ARRAY [1..iProductRecipeArrayQty, 1..iStnQty] OF DSPnpAgitationParameter;

	END_VAR

R_TRIG1(CLK:=bSavePb , Q=> );
R_TRIG2(CLK:=bPnpBusy , Q=> );

IF NOT bPnpBusy THEN
	iStep := 3;
END_IF


IF (iBufferRecipe <> iRecipeStore) OR (iBufferStnID <> iStationID_HMI) THEN
	iStep := 4;
END_IF


IF R_TRIG1.Q THEN
	iStep := 1;
END_IF

IF R_TRIG2.Q THEN
	iStep := 2;
END_IF


CASE iStep OF

0:
bSaveInd	:= FALSE;


1:

	IF iRecipeStore > 0 AND iRecipeStore <= iProductRecipeArrayQty AND iStationID_HMI > 0 AND iStationID_HMI <= iStnQty AND  bAgitationEn THEN

		DSArArmRepeatParaStore[iRecipeStore, iStationID_HMI] := DS_ArmRepeatPara_HMI;
		iBufferRecipe := iRecipeStore;
		iBufferStnID := iStationID_HMI;
		bSaveInd := TRUE;
		iStep := 0;
	END_IF

2:

	IF iRecipeCall >  0 AND iRecipeCall <=  iProductRecipeArrayQty  THEN

		DS_ArmRepeatOut_Pick.lrAgitationTopPosition				:= DSArArmRepeatParaStore[iRecipeCall, iPickNo].lrAgitationTopPosition;
		DS_ArmRepeatOut_Pick.lrAgitationBtmPosition				:= DSArArmRepeatParaStore[iRecipeCall, iPickNo].lrAgitationBtmPosition;
		DS_ArmRepeatOut_Pick.lrAgitationSpeed						:= DSArArmRepeatParaStore[iRecipeCall, iPickNo].lrAgitationSpeed;
		DS_ArmRepeatOut_Pick.lrAgitationSpeedAcc					:= DSArArmRepeatParaStore[iRecipeCall, iPickNo].lrAgitationSpeedAcc;
		DS_ArmRepeatOut_Pick.lrAgitationSpeedDcc					:= DSArArmRepeatParaStore[iRecipeCall, iPickNo].lrAgitationSpeedDcc;
		DS_ArmRepeatOut_Pick.iRepeatUpDownCycle 				:= DSArArmRepeatParaStore[iRecipeCall, iPickNo].iRepeatUpDownCycle;
		DS_ArmRepeatOut_Pick.bPickRepeatStnEnable 				:= DSArArmRepeatParaStore[iRecipeCall, iPickNo].bPickRepeatStnEnable;
		DS_ArmRepeatOut_Pick.bTransferRepeatStnEnable 			:= DSArArmRepeatParaStore[iRecipeCall, iPickNo].bTransferRepeatStnEnable;
		DS_ArmRepeatOut_Pick.bSearchFinish						:= TRUE;

		DS_ArmRepeatOut_Transfer.lrAgitationTopPosition				:= DSArArmRepeatParaStore[iRecipeCall, iTransferNo].lrAgitationTopPosition;
		DS_ArmRepeatOut_Transfer.lrAgitationBtmPosition				:= DSArArmRepeatParaStore[iRecipeCall, iTransferNo].lrAgitationBtmPosition;
		DS_ArmRepeatOut_Transfer.lrAgitationSpeed					:= DSArArmRepeatParaStore[iRecipeCall, iTransferNo].lrAgitationSpeed;
		DS_ArmRepeatOut_Transfer.lrAgitationSpeedAcc				:= DSArArmRepeatParaStore[iRecipeCall, iTransferNo].lrAgitationSpeedAcc;
		DS_ArmRepeatOut_Transfer.lrAgitationSpeedDcc				:= DSArArmRepeatParaStore[iRecipeCall, iTransferNo].lrAgitationSpeedDcc;
		DS_ArmRepeatOut_Transfer.iRepeatUpDownCycle 			:= DSArArmRepeatParaStore[iRecipeCall, iTransferNo].iRepeatUpDownCycle;
		DS_ArmRepeatOut_Transfer.bPickRepeatStnEnable 			:= DSArArmRepeatParaStore[iRecipeCall, iTransferNo].bPickRepeatStnEnable;
		DS_ArmRepeatOut_Transfer.bTransferRepeatStnEnable 		:= DSArArmRepeatParaStore[iRecipeCall, iTransferNo].bTransferRepeatStnEnable;
		DS_ArmRepeatOut_Transfer.bSearchFinish					:= TRUE;

	END_IF
(*
		IF iPickNo <> 0 THEN
			DS_ArmRepeatOut.bPickRepeatStnEnable		:= DSArArmRepeatParaStore[iRecipeCall].ARbPickRepeatStnEnable[iPickNo];
		ELSE
			DS_ArmRepeatOut.bPickRepeatStnEnable		:= FALSE;
		END_IF

		IF iTransferNo <>0 THEN
			DS_ArmRepeatOut.bTransferRepeatStnEnable 	:= DSArArmRepeatParaStore[iRecipeCall].ARbTransferRepeatStnEnable[iTransferNo];
		ELSE
			DS_ArmRepeatOut.bTransferRepeatStnEnable	:= FALSE;
		END_IF
	END_IF
*)

3:
		DS_ArmRepeatOut_Pick := DS_ArmRepeatOut_Empty;
		DS_ArmRepeatOut_Transfer := DS_ArmRepeatOut_Empty;

		iStep := 0;

4:
		DS_ArmRepeatPara_HMI := DSArArmRepeatParaStore[iRecipeStore, iStationID_HMI ];
		iBufferRecipe := iRecipeStore;
		iBufferStnID := iStationID_HMI;
		iStep := 0;


END_CASE


IF NOT bAgitationEn THEN

	DSArArmRepeatParaStore := DSArArmRepeatParaEmpty;
END_IF

END_FUNCTION_BLOCK

// ---- POUs/MainProgram/AutoArmCtrl/PnpMapping_Arm1.TcPOU
PROGRAM PnpMapping_Arm1
VAR

	LeeTest: BOOL;
	LeeTestPnpStart: BOOL;
	LeeTestPSN: INT;
	LeeTestTSN: INT;

END_VAR

(*Arm 1*)
(*Loading*)
		IF ARDSGnrFeedArmPnpParameter[1].iPickStationNo = ARiLdStnID[1] THEN
		ARbDownPickCondition[1]		:=     (
										(bCallRTB_CallOK AND bMTBWriteDoneFlag AND ARDsStnSeqProcessCtrl[0].Out_bProcessCompleted)
										OR
										(bCallRTB_NoTrackerInfo AND bTrackerStartEN AND ARDsStnSeqProcessCtrl[0].Out_bProcessCompleted)
										OR
										(NOT bTimeOptimizeDisable AND ARDsStnSeqProcessCtrl[0].Out_bProcessCompleted)
										)
										AND
										AR2sDSCv_LdConfirmBasketInfo[1,4].iProductRecipeNo >0;
		END_IF

		IF ARDSGnrFeedArmPnpParameter[1].iTransferStationNo = ARiLdStnID[1] THEN
		ARbDownTransferCondition[1]		:=    FALSE;
		END_IF

(*Station 1*)
		IF ARDSGnrFeedArmPnpParameter[1].iPickStationNo = 1 THEN
		ARbDownPickCondition[1]		:=    ARbStationProcessCompletedFlag[1] (*AND ((bArmSlowPullUpCFM AND NOT bStnLiftoutMechanismBypass) OR bStnLiftoutMechanismBypass )*) ;
		END_IF

		IF ARDSGnrFeedArmPnpParameter[1].iTransferStationNo = 1 THEN
		ARbDownTransferCondition[1]		:=    TRUE;
		END_IF

(*Station 2*)
		IF ARDSGnrFeedArmPnpParameter[1].iPickStationNo = 2 THEN
		ARbDownPickCondition[1]		:=    ARbStationProcessCompletedFlag[2] (*AND ((bArmSlowPullUpCFM AND NOT bStnLiftoutMechanismBypass) OR bStnLiftoutMechanismBypass )*) ;
		END_IF

		IF ARDSGnrFeedArmPnpParameter[1].iTransferStationNo = 2 THEN
		ARbDownTransferCondition[1]		:=    TRUE;
		END_IF

(*Station 3*)
		IF ARDSGnrFeedArmPnpParameter[1].iPickStationNo = 3 THEN
		ARbDownPickCondition[1]		:=    ARbStationProcessCompletedFlag[3] (*AND ((bArmSlowPullUpCFM AND NOT bStnLiftoutMechanismBypass) OR bStnLiftoutMechanismBypass )*) ;
		END_IF

		IF ARDSGnrFeedArmPnpParameter[1].iTransferStationNo = 3 THEN
		ARbDownTransferCondition[1]		:=    TRUE;
		END_IF

(*Station 4*)
		IF ARDSGnrFeedArmPnpParameter[1].iPickStationNo = 4 THEN
		ARbDownPickCondition[1]		:=    ARbStationProcessCompletedFlag[4] (*AND ((bArmSlowPullUpCFM AND NOT bStnLiftoutMechanismBypass) OR bStnLiftoutMechanismBypass )*) ;
		END_IF

		IF ARDSGnrFeedArmPnpParameter[1].iTransferStationNo = 4 THEN
		ARbDownTransferCondition[1]		:=    TRUE;
		END_IF

(*Station 5*)
		IF ARDSGnrFeedArmPnpParameter[1].iPickStationNo = 5 THEN
		ARbDownPickCondition[1]		:=    ARbStationProcessCompletedFlag[5] (*AND ((bArmSlowPullUpCFM AND NOT bStnLiftoutMechanismBypass) OR bStnLiftoutMechanismBypass )*) ;
		END_IF

		IF ARDSGnrFeedArmPnpParameter[1].iTransferStationNo = 5 THEN
		ARbDownTransferCondition[1]		:=    TRUE;
		END_IF

(*Station 6*)
		IF ARDSGnrFeedArmPnpParameter[1].iPickStationNo = 6 THEN
		ARbDownPickCondition[1]		:=    ARbStationProcessCompletedFlag[6] (*AND ((bArmSlowPullUpCFM AND NOT bStnLiftoutMechanismBypass) OR bStnLiftoutMechanismBypass )*) ;
		END_IF

		IF ARDSGnrFeedArmPnpParameter[1].iTransferStationNo = 6 THEN
		ARbDownTransferCondition[1]		:=    TRUE;
		END_IF

(*Station 7*)
		IF ARDSGnrFeedArmPnpParameter[1].iPickStationNo = 7 THEN
		ARbDownPickCondition[1]		:=    ARbStationProcessCompletedFlag[7] (*AND ((bArmSlowPullUpCFM AND NOT bStnLiftoutMechanismBypass) OR bStnLiftoutMechanismBypass )*) ;
		END_IF

		IF ARDSGnrFeedArmPnpParameter[1].iTransferStationNo = 7 THEN
		ARbDownTransferCondition[1]		:=    TRUE;
		END_IF

(*Station 8*)
		IF ARDSGnrFeedArmPnpParameter[1].iPickStationNo = 8 THEN
		ARbDownPickCondition[1]		:=    ARbStationProcessCompletedFlag[8] (*AND ((bArmSlowPullUpCFM AND NOT bStnLiftoutMechanismBypass) OR bStnLiftoutMechanismBypass )*) ;
		END_IF

		IF ARDSGnrFeedArmPnpParameter[1].iTransferStationNo = 8 THEN
		ARbDownTransferCondition[1]		:=    TRUE;
		END_IF

(*Station 9*)
		IF ARDSGnrFeedArmPnpParameter[1].iPickStationNo = 9 THEN
		ARbDownPickCondition[1]		:=    ARbStationProcessCompletedFlag[9] AND ((bArmSlowPullUpCFM AND NOT bStnLiftoutMechanismBypass) OR bStnLiftoutMechanismBypass ) ;
		END_IF

		IF ARDSGnrFeedArmPnpParameter[1].iTransferStationNo = 9 THEN
		ARbDownTransferCondition[1]		:=    TRUE;
		END_IF

(*Station 10*)
		IF ARDSGnrFeedArmPnpParameter[1].iPickStationNo = 10 THEN
		ARbDownPickCondition[1]		:=    ARbStationProcessCompletedFlag[10] (*AND ((bArmSlowPullUpCFM AND NOT bStnLiftoutMechanismBypass) OR bStnLiftoutMechanismBypass )*) ;
		END_IF

		IF ARDSGnrFeedArmPnpParameter[1].iTransferStationNo = 10 THEN
		ARbDownTransferCondition[1]		:=    TRUE;
		END_IF

(*Station 11*)
		IF ARDSGnrFeedArmPnpParameter[1].iPickStationNo = 11 THEN
		ARbDownPickCondition[1]		:=    ARbStationProcessCompletedFlag[11] AND ((bArmSlowPullUpCFM AND NOT bStnLiftoutMechanismBypass) OR bStnLiftoutMechanismBypass ) ;
		END_IF

		IF ARDSGnrFeedArmPnpParameter[1].iTransferStationNo = 11 THEN
		ARbDownTransferCondition[1]		:=    TRUE;
		END_IF

(*Station 12*)
		IF ARDSGnrFeedArmPnpParameter[1].iPickStationNo = 12 THEN
		ARbDownPickCondition[1]		:=    ARbStationProcessCompletedFlag[12] AND ((bArmSlowPullUpCFM AND NOT bStnLiftoutMechanismBypass) OR bStnLiftoutMechanismBypass ) ;
		END_IF

		IF ARDSGnrFeedArmPnpParameter[1].iTransferStationNo = 12 THEN
		ARbDownTransferCondition[1]		:=    TRUE;
		END_IF

(*Unloading*)
		IF ARDSGnrFeedArmPnpParameter[1].iPickStationNo = ARiUldStnID[1] (*OR  ARDSGnrFeedArmPnpParameter[1].iPickStationNo = ARiUldStnID[2]*) THEN
		ARbDownPickCondition[1]		:=    FALSE;
		END_IF

		IF ARDSGnrFeedArmPnpParameter[1].iTransferStationNo = ARiUldStnID[1] (*OR  ARDSGnrFeedArmPnpParameter[1].iTransferStationNo = ARiUldStnID[2]*) THEN
		ARbDownTransferCondition[1]		:=    TRUE;
		END_IF

(*Not in Station Range*)
		IF ARDSGnrFeedArmPnpParameter[1].iPickStationNo < 1 OR (ARDSGnrFeedArmPnpParameter[1].iPickStationNo > iStnQty AND ARDSGnrFeedArmPnpParameter[1].iPickStationNo <> ARiLdStnID[1]) THEN
		ARbDownPickCondition[1]		:=    FALSE;
		END_IF

		IF ARDSGnrFeedArmPnpParameter[1].iTransferStationNo < 1 OR (ARDSGnrFeedArmPnpParameter[1].iTransferStationNo > iStnQty AND
		( ARDSGnrFeedArmPnpParameter[1].iTransferStationNo <> ARiUldStnID[1] (*ARiLdStnID[1]*) (*AND ARDSGnrFeedArmPnpParameter[1].iTransferStationNo <> ARiUldStnID[2]*) )) THEN
		ARbDownTransferCondition[1]		:=    FALSE;
		END_IF

(*
IF bLdPnpStart THEN

ARbPnPStart[1]				:=   TRUE 	;
ARiPickStnNo[1]				:=    79	;
ARiTransferStnNo[1]			:=    1	;
ARbDownPickCondition[1]		:=    ( bMTBWriteDoneFlag OR bRecipeTimeBlockTrackerEN OR TRUE) AND LdEnable	;
ARbDownTransferCondition[1]	:=    TRUE	;


ELSIF bStn1PnpStart THEN

ARbPnPStart[1]				:=    TRUE	;
ARiPickStnNo[1]				:=    1	;
ARiTransferStnNo[1]			:=    2	;
ARbDownPickCondition[1]		:=    ARDsStnSeqProcessCtrl[1].Out_bProcessCompleted	;
ARbDownTransferCondition[1]	:=    TRUE	;


ELSIF bStn2PnpStart THEN

ARbPnPStart[1]				:=    TRUE	;
ARiPickStnNo[1]				:=    2	;
ARiTransferStnNo[1]			:=    3	;
ARbDownPickCondition[1]		:=    ARDsStnSeqProcessCtrl[2].Out_bProcessCompleted	;
ARbDownTransferCondition[1]	:=    TRUE	;


ELSIF bStn3PnpStart THEN

ARbPnPStart[1]				:=    TRUE	;
ARiPickStnNo[1]				:=    3	;
ARiTransferStnNo[1]			:=    4	;
ARbDownPickCondition[1]		:=    ARDsStnSeqProcessCtrl[3].Out_bProcessCompleted	;
ARbDownTransferCondition[1]	:=    TRUE	;


ELSIF bStn4PnpStart THEN

ARbPnPStart[1]				:=    TRUE	;
ARiPickStnNo[1]				:=    4	;
ARiTransferStnNo[1]			:=    5	;
ARbDownPickCondition[1]		:=    ARDsStnSeqProcessCtrl[4].Out_bProcessCompleted	;
ARbDownTransferCondition[1]	:=    TRUE	;


ELSIF bStn5PnpStart THEN

ARbPnPStart[1]				:=    TRUE	;
ARiPickStnNo[1]				:=    6	;
ARiTransferStnNo[1]			:=    81	;
ARbDownPickCondition[1]		:=    ARDsStnSeqProcessCtrl[5].Out_bProcessCompleted	;
ARbDownTransferCondition[1]	:=    TRUE	;

ELSIF LeeTest THEN

	ARbPnPStart[1]				:=    LeeTestPnpStart	;
	ARiPickStnNo[1]				:=    LeeTestPSN	;
	ARiTransferStnNo[1]			:=    LeeTestTSN	;
	ARbDownPickCondition[1]		:=    TRUE	;
	ARbDownTransferCondition[1]	:=    TRUE	;
	sStatusMessage;

ELSE

	ARbPnPStart[1]				:=    FALSE	;
	ARiPickStnNo[1]				:=    0	;
	ARiTransferStnNo[1]			:=    0	;
	ARbDownPickCondition[1]		:=    FALSE	;
	ARbDownTransferCondition[1]	:=    FALSE	;

END_IF
*)

ARbPickMidDownStnEn[1]		:= FALSE	;
ARbPickMidDownStnEn[2]		:= FALSE	;
ARbPickMidDownStnEn[3]		:= FALSE	;
ARbPickMidDownStnEn[4]		:= FALSE	;
ARbPickMidDownStnEn[5]		:= FALSE	;
ARbPickMidDownStnEn[6]		:= FALSE	;
ARbPickMidDownStnEn[7]		:= FALSE	; (*TRUE AND NOT bStnLiftoutMechanismBypass;*)
ARbPickMidDownStnEn[8]		:= FALSE	;
ARbPickMidDownStnEn[9]		:= TRUE AND NOT bStnLiftoutMechanismBypass	;
ARbPickMidDownStnEn[10]		:= FALSE	;
ARbPickMidDownStnEn[11]		:= FALSE	;
ARbPickMidDownStnEn[12]		:= FALSE	;

ARbTransferMidDownStnEn[1]	:= FALSE	;
ARbTransferMidDownStnEn[2]	:= FALSE	;
ARbTransferMidDownStnEn[3]	:= FALSE	;
ARbTransferMidDownStnEn[4]	:= FALSE	;
ARbTransferMidDownStnEn[5]	:= FALSE	;
ARbTransferMidDownStnEn[6]	:= FALSE	;
ARbTransferMidDownStnEn[7]	:= FALSE	;
ARbTransferMidDownStnEn[8]	:= FALSE	;
ARbTransferMidDownStnEn[9]	:= FALSE	;
ARbTransferMidDownStnEn[10]	:= FALSE	;
ARbTransferMidDownStnEn[11]	:= FALSE	;
ARbTransferMidDownStnEn[12]	:= FALSE	;

ARiStationDippingTime[1]		:= ARiStnDippingTimeSV[1]	;
ARiStationDippingTime[2]		:= ARiStnDippingTimeSV[2]	;
ARiStationDippingTime[3]		:= ARiStnDippingTimeSV[3]	;
ARiStationDippingTime[4]		:= ARiStnDippingTimeSV[4]	;
ARiStationDippingTime[5]		:= ARiStnDippingTimeSV[5]	;
ARiStationDippingTime[6]		:= ARiStnDippingTimeSV[6]	;
ARiStationDippingTime[7]		:= ARiStnDippingTimeSV[7]	;
ARiStationDippingTime[8]		:= ARiStnDippingTimeSV[8]	;
ARiStationDippingTime[9]		:= ARiStnDippingTimeSV[9]	;
ARiStationDippingTime[10]		:= ARiStnDippingTimeSV[10];
ARiStationDippingTime[11]		:= ARiStnDippingTimeSV[11];
ARiStationDippingTime[12]		:= ARiStnDippingTimeSV[12];

(********************Output************************)
(*Top Triggering*)
bArm1VertLD1Up_15 			:= bMoveTop;

(*Vert Triggering*)
bArm1VertLD1Down_05 		:= ARbMoveLdDown[1];
bArm1VertULD1Down_05 		:= ARbMoveUldDown[1];

bArm1VertStn1Down_05		:= ARbMoveStnDown[1];
bArm1VertStn2Down_05		:= ARbMoveStnDown[2];
bArm1VertStn3Down_05		:= ARbMoveStnDown[3];
bArm1VertStn4Down_05		:= ARbMoveStnDown[4];
bArm1VertStn5Down_05		:= ARbMoveStnDown[5];
bArm1VertStn6Down_05		:= ARbMoveStnDown[6];
bArm1VertStn7Down_05		:= ARbMoveStnDown[7];
bArm1VertStn8Down_05		:= ARbMoveStnDown[8];
bArm1VertStn9Down_05		:= ARbMoveStnDown[9];
bArm1VertStn10Down_05		:= ARbMoveStnDown[10];
bArm1VertStn11Down_05		:= ARbMoveStnDown[11];
bArm1VertStn12Down_05		:= ARbMoveStnDown[12];

bArm1VertStn1SpSlanted_05 	:= ARbMoveStnMidDown[1];
bArm1VertStn2SpSlanted_05 	:= ARbMoveStnMidDown[2];
bArm1VertStn3SpSlanted_05 	:= ARbMoveStnMidDown[3];
bArm1VertStn4SpSlanted_05 	:= ARbMoveStnMidDown[4];
bArm1VertStn5SpSlanted_05 	:= ARbMoveStnMidDown[5];
bArm1VertStn6SpSlanted_05 	:= ARbMoveStnMidDown[6];
bArm1VertStn7SpSlanted_05 	:= ARbMoveStnMidDown[7];
bArm1VertStn8SpSlanted_05 	:= ARbMoveStnMidDown[8];
bArm1VertStn9SpSlanted_05 	:= ARbMoveStnMidDown[9];
bArm1VertStn10SpSlanted_05 	:= ARbMoveStnMidDown[10];
bArm1VertStn11SpSlanted_05 	:= ARbMoveStnMidDown[11];
bArm1VertStn12SpSlanted_05 	:= ARbMoveStnMidDown[12];


(*Hook Triggering*)
bArm1HorzLD1Hook_05 		:= ARbMoveLdHook[1];
bArm1HorzLD1Unhook_05		:= ARbMoveLdUnhook[1];

bArm1HorzStn1Hook_05 		:= ARbMoveStnHook[1];
bArm1HorzStn2Hook_05 		:= ARbMoveStnHook[2];
bArm1HorzStn3Hook_05 		:= ARbMoveStnHook[3];
bArm1HorzStn4Hook_05 		:= ARbMoveStnHook[4];
bArm1HorzStn5Hook_05 		:= ARbMoveStnHook[5];
bArm1HorzStn6Hook_05 		:= ARbMoveStnHook[6];
bArm1HorzStn7Hook_05 		:= ARbMoveStnHook[7];
bArm1HorzStn8Hook_05 		:= ARbMoveStnHook[8];
bArm1HorzStn9Hook_05 		:= ARbMoveStnHook[9];
bArm1HorzStn10Hook_05 		:= ARbMoveStnHook[10];
bArm1HorzStn11Hook_05 		:= ARbMoveStnHook[11];
bArm1HorzStn12Hook_05 		:= ARbMoveStnHook[12];

(*Unhook Triggering*)
bArm1HorzULD1Hook_05 		:= ARbMoveUldHook[1];
bArm1HorzULD1Unhook_05 		:= ARbMoveUldUnhook[1];

bArm1HorzStn1Unhook_05 		:= ARbMoveStnUnhook[1];
bArm1HorzStn2Unhook_05 		:= ARbMoveStnUnhook[2];
bArm1HorzStn3Unhook_05 		:= ARbMoveStnUnhook[3];
bArm1HorzStn4Unhook_05 		:= ARbMoveStnUnhook[4];
bArm1HorzStn5Unhook_05 		:= ARbMoveStnUnhook[5];
bArm1HorzStn6Unhook_05 		:= ARbMoveStnUnhook[6];
bArm1HorzStn7Unhook_05 		:= ARbMoveStnUnhook[7];
bArm1HorzStn8Unhook_05 		:= ARbMoveStnUnhook[8];
bArm1HorzStn9Unhook_05 		:= ARbMoveStnUnhook[9];
bArm1HorzStn10Unhook_05 	:= ARbMoveStnUnhook[10];
bArm1HorzStn11Unhook_05		:= ARbMoveStnUnhook[11];
bArm1HorzStn12Unhook_05 	:= ARbMoveStnUnhook[12];


ARDSArmCtrl[1].AR3sbPositionCfm[1,1,1]		:= ARDSArmCtrl[1].AR3sbPositionCfm[2,1,1]; (*STN1*)
ARDSArmCtrl[1].AR3sbPositionCfm[1,2,1] 		:= ARDSArmCtrl[1].AR3sbPositionCfm[2,1,1]; (*STN2*)
ARDSArmCtrl[1].AR3sbPositionCfm[1,3,1]		:= ARDSArmCtrl[1].AR3sbPositionCfm[2,1,1]; (*STN3*)
ARDSArmCtrl[1].AR3sbPositionCfm[1,4,1] 		:= ARDSArmCtrl[1].AR3sbPositionCfm[2,1,1]; (*STN4*)
ARDSArmCtrl[1].AR3sbPositionCfm[1,5,1]		:= ARDSArmCtrl[1].AR3sbPositionCfm[2,1,1]; (*STN5*)
ARDSArmCtrl[1].AR3sbPositionCfm[1,6,1] 		:= ARDSArmCtrl[1].AR3sbPositionCfm[2,1,1]; (*STN6*)
ARDSArmCtrl[1].AR3sbPositionCfm[1,7,1]		:= ARDSArmCtrl[1].AR3sbPositionCfm[2,1,1]; (*STN7*)
ARDSArmCtrl[1].AR3sbPositionCfm[1,8,1] 		:= ARDSArmCtrl[1].AR3sbPositionCfm[2,1,1]; (*STN8*)
ARDSArmCtrl[1].AR3sbPositionCfm[1,9,1]		:= ARDSArmCtrl[1].AR3sbPositionCfm[2,1,1]; (*STN9*)
ARDSArmCtrl[1].AR3sbPositionCfm[1,10,1]		:= ARDSArmCtrl[1].AR3sbPositionCfm[2,1,1]; (*STN10*)
ARDSArmCtrl[1].AR3sbPositionCfm[1,11,1]		:= ARDSArmCtrl[1].AR3sbPositionCfm[2,1,1]; (*STN11*)
ARDSArmCtrl[1].AR3sbPositionCfm[1,12,1]		:= ARDSArmCtrl[1].AR3sbPositionCfm[2,1,1]; (*STN12*)
ARDSArmCtrl[1].AR3sbPositionCfm[3,1,1]		:= ARDSArmCtrl[1].AR3sbPositionCfm[2,1,1]; (*ULD1*)
ARDSArmCtrl[1].AR3sbPositionCfm[3,2,1]		:= ARDSArmCtrl[1].AR3sbPositionCfm[2,1,1]; (*ULD2*)


ARDSStnInterlock[1].ARbArmUpInterlock[1]		:= bArm1LdUpInterlockOK;
ARDSStnInterlock[1].ARbArmUpInterlock[2]		:= bArm1LdUpInterlockOK;
ARDSStnInterlock[1].ARbArmUpInterlock[3]		:= bArm1LdUpInterlockOK;
ARDSStnInterlock[1].ARbArmUpInterlock[4]		:= bArm1LdUpInterlockOK;
ARDSStnInterlock[1].ARbArmUpInterlock[5]		:= bArm1LdUpInterlockOK;
ARDSStnInterlock[1].ARbArmUpInterlock[6]		:= bArm1LdUpInterlockOK;
ARDSStnInterlock[1].ARbArmUpInterlock[7]		:= bArm1LdUpInterlockOK;
ARDSStnInterlock[1].ARbArmUpInterlock[8]		:= bArm1LdUpInterlockOK;
ARDSStnInterlock[1].ARbArmUpInterlock[9]		:= bArm1LdUpInterlockOK;
ARDSStnInterlock[1].ARbArmUpInterlock[10]		:= bArm1LdUpInterlockOK;
ARDSStnInterlock[1].ARbArmUpInterlock[11]		:= bArm1LdUpInterlockOK;
ARDSStnInterlock[1].ARbArmUpInterlock[12]		:= bArm1LdUpInterlockOK;

ARDSStnInterlock[2].ARbArmUpInterlock[1]		:= bArm2LdUpInterlockOK;
ARDSStnInterlock[2].ARbArmUpInterlock[2]		:= bArm2LdUpInterlockOK;
ARDSStnInterlock[2].ARbArmUpInterlock[3]		:= bArm2LdUpInterlockOK;
ARDSStnInterlock[2].ARbArmUpInterlock[4]		:= bArm2LdUpInterlockOK;
ARDSStnInterlock[2].ARbArmUpInterlock[5]		:= bArm2LdUpInterlockOK;
ARDSStnInterlock[2].ARbArmUpInterlock[6]		:= bArm2LdUpInterlockOK;
ARDSStnInterlock[2].ARbArmUpInterlock[7]		:= bArm2LdUpInterlockOK;
ARDSStnInterlock[2].ARbArmUpInterlock[8]		:= bArm2LdUpInterlockOK;
ARDSStnInterlock[2].ARbArmUpInterlock[9]		:= bArm2LdUpInterlockOK;
ARDSStnInterlock[2].ARbArmUpInterlock[10]		:= bArm2LdUpInterlockOK;
ARDSStnInterlock[2].ARbArmUpInterlock[11]		:= bArm2LdUpInterlockOK;
ARDSStnInterlock[2].ARbArmUpInterlock[12]		:= bArm2LdUpInterlockOK;

END_PROGRAM

// ---- POUs/MainProgram/AutoArmCtrl/PnPstorageMemory_Arm.TcPOU
PROGRAM PnPstorageMemory_Arm
VAR
	fbGnrProductRecipeMemory_Main: fbV2_GnrProductRecipeMemory;
	tProductRecipeClearPb : TON;
END_VAR

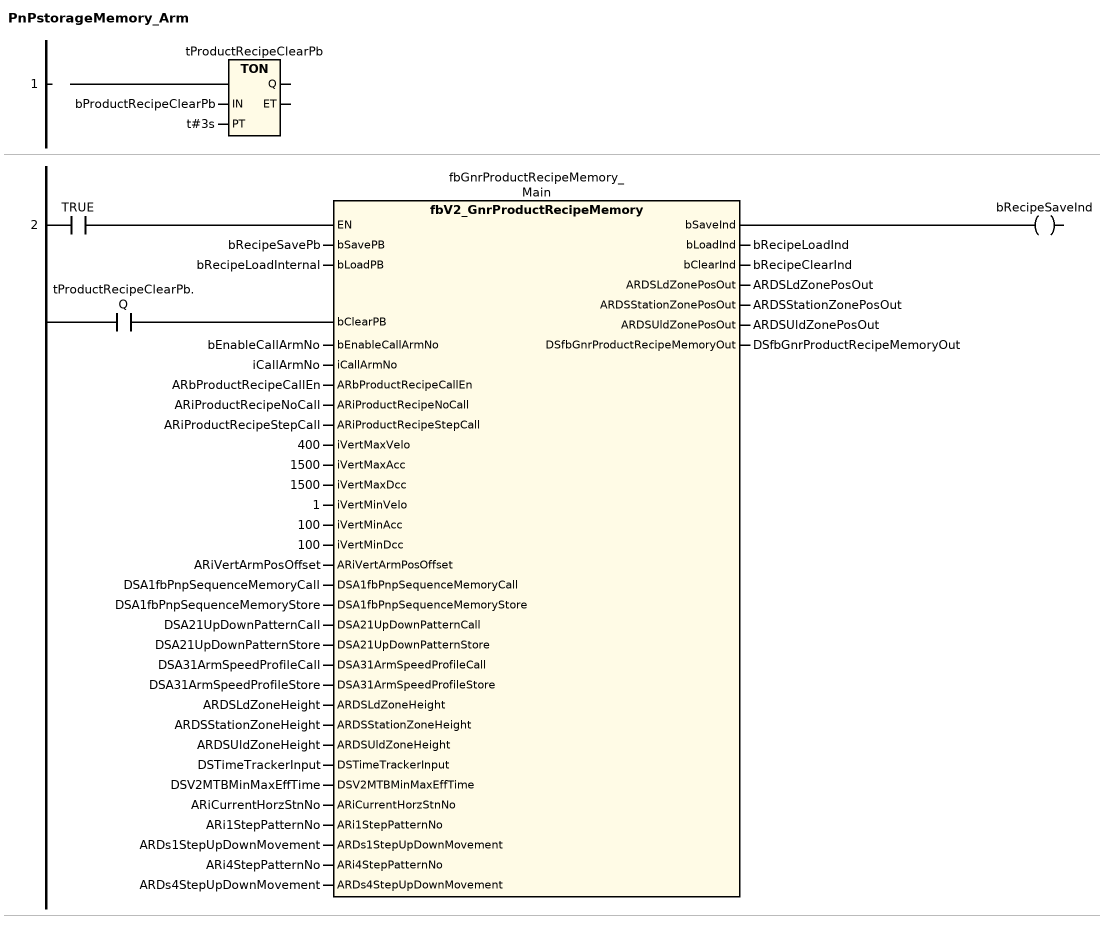
// NETWORK 1
tProductRecipeClearPb(IN := bProductRecipeClearPb, PT := t#3s); // TON

// NETWORK 2
fbGnrProductRecipeMemory_Main(
    bSavePB := bRecipeSavePb,
    bLoadPB := bRecipeLoadInternal,
    bClearPB := tProductRecipeClearPb.Q,
    bEnableCallArmNo := bEnableCallArmNo,
    iCallArmNo := iCallArmNo,
    ARbProductRecipeCallEn := ARbProductRecipeCallEn,
    ARiProductRecipeNoCall := ARiProductRecipeNoCall,
    ARiProductRecipeStepCall := ARiProductRecipeStepCall,
    iVertMaxVelo := 400,
    iVertMaxAcc := 1500,
    iVertMaxDcc := 1500,
    iVertMinVelo := 1,
    iVertMinAcc := 100,
    iVertMinDcc := 100,
    ARiVertArmPosOffset := ARiVertArmPosOffset,
    DSA1fbPnpSequenceMemoryCall := DSA1fbPnpSequenceMemoryCall,
    DSA1fbPnpSequenceMemoryStore := DSA1fbPnpSequenceMemoryStore,
    DSA21UpDownPatternCall := DSA21UpDownPatternCall,
    DSA21UpDownPatternStore := DSA21UpDownPatternStore,
    DSA31ArmSpeedProfileCall := DSA31ArmSpeedProfileCall,
    DSA31ArmSpeedProfileStore := DSA31ArmSpeedProfileStore,
    ARDSLdZoneHeight := ARDSLdZoneHeight,
    ARDSStationZoneHeight := ARDSStationZoneHeight,
    ARDSUldZoneHeight := ARDSUldZoneHeight,
    DSTimeTrackerInput := DSTimeTrackerInput,
    DSV2MTBMinMaxEffTime := DSV2MTBMinMaxEffTime,
    ARiCurrentHorzStnNo := ARiCurrentHorzStnNo,
    ARi1StepPatternNo := ARi1StepPatternNo,
    ARDs1StepUpDownMovement := ARDs1StepUpDownMovement,
    ARi4StepPatternNo := ARi4StepPatternNo,
    ARDs4StepUpDownMovement := ARDs4StepUpDownMovement,
    bLoadInd => bRecipeLoadInd,
    bClearInd => bRecipeClearInd,
    ARDSLdZonePosOut => ARDSLdZonePosOut,
    ARDSStationZonePosOut => ARDSStationZonePosOut,
    ARDSUldZonePosOut => ARDSUldZonePosOut,
    DSfbGnrProductRecipeMemoryOut => DSfbGnrProductRecipeMemoryOut); // fbV2_GnrProductRecipeMemory
bRecipeSaveInd := fbGnrProductRecipeMemory_Main.bSaveInd;

END_PROGRAM

// ---- FBs/B_JKS_NewFB_V2/FBP-ArmRelated/fbV2_GnrProductRecipeMemory.TcPOU
FUNCTION_BLOCK fbV2_GnrProductRecipeMemory

VAR_INPUT
	bSavePB  : BOOL;
	bLoadPB  : BOOL;
	bClearPB : BOOL;
	bEnableCallArmNo : BOOL;
	iCallArmNo : INT;

	ARbProductRecipeCallEn(*ARbArmPnpSequenceStorageCall*) 	: ARRAY [0..iStnQty] OF BOOL;
	ARiProductRecipeNoCall(*ARiPnpSequenceNoCall*) 			: ARRAY [0..iStnQty] OF INT;
	ARiProductRecipeStepCall(*ARiPnpSequenceStepCall*) 		: ARRAY [0..iStnQty] OF INT;


	iVertMaxVelo : INT;
	iVertMaxAcc : INT;
	iVertMaxDcc : INT;
	iVertMinVelo : INT;
	iVertMinAcc : INT;
	iVertMinDcc : INT;

END_VAR
VAR_OUTPUT

	bSaveInd : BOOL;
	bLoadInd : BOOL;
	bClearInd : BOOL;

	ARDSLdZonePosOut			: ARRAY [0..iLdStnQty] OF DSA32_StationZonePosOut;
	ARDSStationZonePosOut 		: ARRAY [0..iStnQty] OF DSA32_StationZonePosOut;
	ARDSUldZonePosOut 			: ARRAY [0..iUldStnQty] OF DSA32_StationZonePosOut;

(*	bCallCompleted : BOOL;*)
(*
	bInvalidProductRecipeNoErrHold(*bInvalidPnpSequenceNoErrHold*) : BOOL;
	bInvalidProductRecipeNoErrPulse(*bInvalidPnpSequenceNoErrPulse*): BOOL;
	bInvalidProductRecipeStepErrHold(*bInvalidPnpSequenceStepErrHold*) : BOOL;
	bInvalidProductRecipeStepErrPulse(*bInvalidPnpSequenceStepErrPulse*): BOOL;
*)
(*
	bCallUpDownPatternMemoryErr : BOOL;
	
 : BOOL;
	bCallPickStationNoErr : BOOL;
	bCallTransferStationNoErr : BOOL;
*)(*
	iCalledProductRecipeNo(*iCalledPnpSequenceNo*) : INT; (*New*)
	iCalledProductRecipeStep(*iCalledPnpSequenceStep*): INT; (*New*)
	sProductRecipeDescription(*sPnpSequenceDescription*) : STRING(50);
(*	DSA1CalledDownPickMovement : DSA1_UpDownMovement;
	DSA1CalledUpPickMovement : DSA1_UpDownMovement;
	DSA1CalledDownTransferMovement : DSA1_UpDownMovement;
	DSA1CalledUpTransferMovement : DSA1_UpDownMovement;
*)


(*Continue Here*)
	DSGnrCalledArmPnpParameter : DSGnr_CalledArmPnpParameter;

	iCallCaseNo : INT;*)

	DSfbGnrProductRecipeMemoryOut : DSV2_fbGnrProductRecipeMemoryOut;

END_VAR

VAR_IN_OUT PERSISTENT

(*	ARiLdStnID : INT;
	ARiUldStnID : INT;
*)(*	ARiArmID : ARRAY [0..iArmQty] OF INT;*)
	ARiVertArmPosOffset : ARRAY [0..iArmQty] OF INT;
	DSA1fbPnpSequenceMemoryCall : DSV2_A1_fbPnpSequenceMemoryCall;
	DSA1fbPnpSequenceMemoryStore : DSV2_A1_fbPnpSequenceMemoryStore;

	DSA21UpDownPatternCall : DSA21_UpDownPatternCall;
	DSA21UpDownPatternStore : DSA21_UpDownPatternStore;

	DSA31ArmSpeedProfileCall : DSA31_ArmSpeedProfileCall;
	DSA31ArmSpeedProfileStore : DSA31_ArmSpeedProfileStore;

	ARDSLdZoneHeight : ARRAY [0..iLdStnQty] OF DSA32_StationZoneHeight;
	ARDSStationZoneHeight : ARRAY [0..iStnQty] OF DSA32_StationZoneHeight;
	ARDSUldZoneHeight : ARRAY [0..iUldStnQty] OF DSA32_StationZoneHeight;

	DSTimeTrackerInput : DSV2_TimeTrackerInput; (*New*)
	DSV2MTBMinMaxEffTime : DSV2_MinMaxEffTime;
	ARiCurrentHorzStnNo						: ARRAY [1..iArmQty] OF INT;
	ARi1StepPatternNo						: ARRAY [1..iArmQty] OF INT;
	ARDs1StepUpDownMovement			: ARRAY [1..iArmQty] OF DSA1_UpDownMovement;
	ARi4StepPatternNo						: ARRAY [1..iArmQty] OF INT;
	ARDs4StepUpDownMovement			: ARRAY [1..iArmQty] OF DSA1_UpDownMovement;


END_VAR

VAR (*PERSISTENT*)

	fbA1PnpSequenceMemory: fbV2_A1_PnpSequenceMemory;
	fbA21UpDownPattern: fbA21_UpDownPattern;
	fbA31ArmSpeedProfileMemory: fbA31_ArmSpeedProfileMemory;
	fbV2A32MachineZoneHeight: fbV2_A32_MachineZoneHeight;


	iPull1StepSFL: INT;
	iPull4StepSFL: INT;
	iBufTransStnNoCheckFL: INT;

	bTransStnFound: BOOL;
	iTransStnID: INT;

	bTransLdStnFound: BOOL;
	iTransLdStnID: INT;

	bTransUldStnFound: BOOL;
	iTransUldStnID: INT;


	iBufPickStnNoCheckFL: INT;

	bPickStnFound: BOOL;
	iPickStnID: INT;

	bPickLdStnFound: BOOL;
	iPickLdStnID: INT;

	bPickUldStnFound: BOOL;
	iPickUldStnID: INT;
	iSSERFL: INT;
END_VAR
VAR
	iProductRecipeNoCall(*iPnpSequenceNoCall*) : INT;
	iProductRecipeStepCall(*iPnpSequenceStepCall*): INT;
	bCallSt: BOOL;

	CallSelfCheckHR: BOOL;
(*	iPreviousPnpSequenceStep(*iPreviousPnpSequenceStep*): INT;*)
	CallSelfCheckRE : R_TRIG;
(*	febInvalidProductRecipeeNo(*febInvalidPnpSequenceNo*) : F_TRIG;
	febInvalidProductRecipeStep(*febInvalidPnpSequenceStep*) : F_TRIG;
*)
	tInvalidProductRecipeNoErrTimer(*tInvalidPnpSequenceNoErrTimer*): TON;
	tInvalidProductRecipeStepErrTimer(*tInvalidPnpSequenceStepErrTimer*): TON;
	rebInvalidProductRecipeNo(*rebInvalidPnpSequenceNo*): R_TRIG;
	rebInvalidProductRecipeStep(*rebInvalidPnpSequenceStep*): R_TRIG;

	reCallCompleted: R_TRIG;
	CallCompletedTimer: TON;

	rebInvalidUpDownPatternMemoryCall: R_TRIG;
	rebInvalidSpeedProfileMemoryCall: R_TRIG;
	rebCallSt: R_TRIG;
	tCallArmSpeedProfileMemoryErrTimer: TON;
	tCallUpDownPatternMemoryErrTimer: TON;

	iBufferPickStationNo: INT;
	iBufferTransferStationNo: INT;

	iBufferDownPickPatternNo: INT;
	iBufferUpPickPatternNo: INT;
	iBufferDownTransferPatternNo: INT;
	iBufferUpTransferPatternNo: INT;

	DSBufferDownPickPattern : DSA21_UpDownPatternMemory;
	DSBufferUpPickPattern : DSA21_UpDownPatternMemory;
	DSBufferDownTransferPattern : DSA21_UpDownPatternMemory;
	DSBufferUpTransferPattern : DSA21_UpDownPatternMemory;

(*	DSBufferDownPickSpdProfile : ARRAY [1..4] OF DSA31_ArmSpeedProfileMemory;
	DSBufferUpPickSpdProfile : ARRAY [1..4] OF DSA31_ArmSpeedProfileMemory;
	DSBufferDownTransferSpdProfile : ARRAY [1..4] OF DSA31_ArmSpeedProfileMemory;
	DSBufferUpTransferSpdProfile : ARRAY [1..4] OF DSA31_ArmSpeedProfileMemory;*)


	bCallStRE: R_TRIG;
	bCallStFE: F_TRIG;
	tCallPickStationNoErrTimer: TON;
	tCallTransferStationNoErrTimer: TON;
	iCallCheck: INT;
	iCalledDataRequestFromStationNo: INT;
	bCalledDataRequestStationFound: BOOL;
	iPull1StepFL: INT;
	iPull4StepFL: INT;
	DSEmptyPnpSequenceMemory : DSV2_A1_PnpSequenceMemory;

END_VAR

(*****************READ  SSER based on ProductRecipeNo and TransferStationNo START****************************)

IF DSV2MTBMinMaxEffTime.iProductRecipeNo > 0 AND DSV2MTBMinMaxEffTime.iProductRecipeNo <= iProductRecipeArrayQty THEN

	DSV2MTBMinMaxEffTime.ARiTransferStationNo 	:= fbA1PnpSequenceMemory.ARDsPnpSequenceMemory[DSV2MTBMinMaxEffTime.iProductRecipeNo].ARiTransferStationNo;
	DSV2MTBMinMaxEffTime.ARiStnSeqRepNo		:= fbA1PnpSequenceMemory.ARDsPnpSequenceMemory[DSV2MTBMinMaxEffTime.iProductRecipeNo].ARiStnSeqRepNo;

END_IF




(*****************READ  SSER based on ProductRecipeNo and TransferStationNo END****************************)


(*[][][][][][][][][][][][][][][][][][][][][][][][][][][][][][][][][][][][][][][][][][][][][][][][][][][][][][][][][][][][][][][][][][][][][][][][][][][][][][][][][][][][][][][][][][][][][][][][][][][]*)
(*Call TimeTracker - Product Recipe Info*)
IF DSTimeTrackerInput.iTimeTrackerProductRecipeNo > 0 AND DSTimeTrackerInput.iTimeTrackerProductRecipeNo <= iProductRecipeArrayQty THEN
DSTimeTrackerInput.ARiCallArmNo 									:= fbA1PnpSequenceMemory.ARDsPnpSequenceMemory[DSTimeTrackerInput.iTimeTrackerProductRecipeNo].ARiCallArmNo;
DSTimeTrackerInput.ARiPickStationNo								:= fbA1PnpSequenceMemory.ARDsPnpSequenceMemory[DSTimeTrackerInput.iTimeTrackerProductRecipeNo].ARiPickStationNo;
DSTimeTrackerInput.ARiStnSeqRepNo 								:= fbA1PnpSequenceMemory.ARDsPnpSequenceMemory[DSTimeTrackerInput.iTimeTrackerProductRecipeNo].ARiStnSeqRepNo;
DSTimeTrackerInput.ARiTransferStationNo 							:= fbA1PnpSequenceMemory.ARDsPnpSequenceMemory[DSTimeTrackerInput.iTimeTrackerProductRecipeNo].ARiTransferStationNo;
DSTimeTrackerInput.iLdGroupNo									:= fbA1PnpSequenceMemory.ARDsPnpSequenceMemory[DSTimeTrackerInput.iTimeTrackerProductRecipeNo].iLdGroupNo;
DSTimeTrackerInput.iUldGroupNo									:= fbA1PnpSequenceMemory.ARDsPnpSequenceMemory[DSTimeTrackerInput.iTimeTrackerProductRecipeNo].iUldGroupNo;

ELSE
DSTimeTrackerInput.ARiCallArmNo 									:= DSEmptyPnpSequenceMemory.ARiCallArmNo;
DSTimeTrackerInput.ARiPickStationNo								:= DSEmptyPnpSequenceMemory.ARiPickStationNo;
DSTimeTrackerInput.ARiStnSeqRepNo 								:= DSEmptyPnpSequenceMemory.ARiStnSeqRepNo;
DSTimeTrackerInput.ARiTransferStationNo 							:= DSEmptyPnpSequenceMemory.ARiTransferStationNo;
DSTimeTrackerInput.iLdGroupNo									:= fbA1PnpSequenceMemory.ARDsPnpSequenceMemory[DSTimeTrackerInput.iTimeTrackerProductRecipeNo].iLdGroupNo;
DSTimeTrackerInput.iUldGroupNo									:= fbA1PnpSequenceMemory.ARDsPnpSequenceMemory[DSTimeTrackerInput.iTimeTrackerProductRecipeNo].iUldGroupNo;
END_IF


(*1 Step UpDownMovement Data Pulling*)
iPull1StepFL := 1;

FOR iPull1StepFL := 1 TO iArmQty DO
	IF iPull1StepFL >=1 AND iPull1StepFL <= iArmQty THEN

			IF ARiCurrentHorzStnNo[iPull1StepFL] >= 1 AND ARiCurrentHorzStnNo[iPull1StepFL] <= iStnQty THEN
			ARDs1StepUpDownMovement[iPull1StepFL].lrZone1StartPos					:= ARDSStationZonePosOut[ARiCurrentHorzStnNo[iPull1StepFL]].lrZone1StartPos - ARiVertArmPosOffset[iPull1StepFL];
			ARDs1StepUpDownMovement[iPull1StepFL].lrZone1EndPos					:= ARDSStationZonePosOut[ARiCurrentHorzStnNo[iPull1StepFL]].lrZone1EndPos - ARiVertArmPosOffset[iPull1StepFL];
			ARDs1StepUpDownMovement[iPull1StepFL].lrZone2StartPos					:= ARDSStationZonePosOut[ARiCurrentHorzStnNo[iPull1StepFL]].lrZone2StartPos - ARiVertArmPosOffset[iPull1StepFL];
			ARDs1StepUpDownMovement[iPull1StepFL].lrZone2EndPos					:= ARDSStationZonePosOut[ARiCurrentHorzStnNo[iPull1StepFL]].lrZone2EndPos - ARiVertArmPosOffset[iPull1StepFL];
			ARDs1StepUpDownMovement[iPull1StepFL].lrZone3StartPos					:= ARDSStationZonePosOut[ARiCurrentHorzStnNo[iPull1StepFL]].lrZone3StartPos - ARiVertArmPosOffset[iPull1StepFL];
			ARDs1StepUpDownMovement[iPull1StepFL].lrZone3EndPos					:= ARDSStationZonePosOut[ARiCurrentHorzStnNo[iPull1StepFL]].lrZone3EndPos - ARiVertArmPosOffset[iPull1StepFL];
			ARDs1StepUpDownMovement[iPull1StepFL].lrZone4StartPos					:= ARDSStationZonePosOut[ARiCurrentHorzStnNo[iPull1StepFL]].lrZone4StartPos - ARiVertArmPosOffset[iPull1StepFL];
			ARDs1StepUpDownMovement[iPull1StepFL].lrZone4EndPos					:= ARDSStationZonePosOut[ARiCurrentHorzStnNo[iPull1StepFL]].lrZone4EndPos - ARiVertArmPosOffset[iPull1StepFL];

			ARDs1StepUpDownMovement[iPull1StepFL].lrMidPos							:= ARDSStationZonePosOut[ARiCurrentHorzStnNo[iPull1StepFL]].lrMidPos;

			ELSE

			iPull1StepSFL := 1;
				FOR iPull1StepSFL := 1 TO iLdStnQty DO
					IF iPull1StepSFL >=1 AND iPull1StepSFL <= iLdStnQty THEN

						(*With Condition*)
						IF ARiCurrentHorzStnNo[iPull1StepFL] = ARiLdStnID[iPull1StepSFL] THEN
						ARDs1StepUpDownMovement[iPull1StepFL].lrZone1StartPos					:= ARDSLdZonePosOut[iPull1StepSFL].lrZone1StartPos - ARiVertArmPosOffset[ARiCurrentHorzStnNo[iPull1StepFL]];
						ARDs1StepUpDownMovement[iPull1StepFL].lrZone1EndPos					:= ARDSLdZonePosOut[iPull1StepSFL].lrZone1EndPos - ARiVertArmPosOffset[ARiCurrentHorzStnNo[iPull1StepFL]];
						ARDs1StepUpDownMovement[iPull1StepFL].lrZone2StartPos					:= ARDSLdZonePosOut[iPull1StepSFL].lrZone2StartPos - ARiVertArmPosOffset[ARiCurrentHorzStnNo[iPull1StepFL]];
						ARDs1StepUpDownMovement[iPull1StepFL].lrZone2EndPos					:= ARDSLdZonePosOut[iPull1StepSFL].lrZone2EndPos - ARiVertArmPosOffset[ARiCurrentHorzStnNo[iPull1StepFL]];
						ARDs1StepUpDownMovement[iPull1StepFL].lrZone3StartPos					:= ARDSLdZonePosOut[iPull1StepSFL].lrZone3StartPos - ARiVertArmPosOffset[ARiCurrentHorzStnNo[iPull1StepFL]];
						ARDs1StepUpDownMovement[iPull1StepFL].lrZone3EndPos					:= ARDSLdZonePosOut[iPull1StepSFL].lrZone3EndPos - ARiVertArmPosOffset[ARiCurrentHorzStnNo[iPull1StepFL]];
						ARDs1StepUpDownMovement[iPull1StepFL].lrZone4StartPos					:= ARDSLdZonePosOut[iPull1StepSFL].lrZone4StartPos - ARiVertArmPosOffset[ARiCurrentHorzStnNo[iPull1StepFL]];
						ARDs1StepUpDownMovement[iPull1StepFL].lrZone4EndPos					:= ARDSLdZonePosOut[iPull1StepSFL].lrZone4EndPos - ARiVertArmPosOffset[ARiCurrentHorzStnNo[iPull1StepFL]];
			
						ARDs1StepUpDownMovement[iPull1StepFL].lrMidPos							:= ARDSLdZonePosOut[iPull1StepSFL].lrMidPos;

						END_IF
					END_IF
				END_FOR

			iPull1StepSFL := 1;
				FOR iPull1StepSFL := 1 TO iUldStnQty DO
					IF iPull1StepSFL >=1 AND iPull1StepSFL <= iUldStnQty THEN


						IF ARiCurrentHorzStnNo[iPull1StepFL] = ARiUldStnID[iPull1StepSFL] THEN
						ARDs1StepUpDownMovement[iPull1StepFL].lrZone1StartPos					:= ARDSUldZonePosOut[iPull1StepSFL].lrZone1StartPos - ARiVertArmPosOffset[iPull1StepFL];
						ARDs1StepUpDownMovement[iPull1StepFL].lrZone1EndPos					:= ARDSUldZonePosOut[iPull1StepSFL].lrZone1EndPos - ARiVertArmPosOffset[iPull1StepFL];
						ARDs1StepUpDownMovement[iPull1StepFL].lrZone2StartPos					:= ARDSUldZonePosOut[iPull1StepSFL].lrZone2StartPos - ARiVertArmPosOffset[iPull1StepFL];
						ARDs1StepUpDownMovement[iPull1StepFL].lrZone2EndPos					:= ARDSUldZonePosOut[iPull1StepSFL].lrZone2EndPos - ARiVertArmPosOffset[iPull1StepFL];
						ARDs1StepUpDownMovement[iPull1StepFL].lrZone3StartPos					:= ARDSUldZonePosOut[iPull1StepSFL].lrZone3StartPos - ARiVertArmPosOffset[iPull1StepFL];
						ARDs1StepUpDownMovement[iPull1StepFL].lrZone3EndPos					:= ARDSUldZonePosOut[iPull1StepSFL].lrZone3EndPos - ARiVertArmPosOffset[iPull1StepFL];
						ARDs1StepUpDownMovement[iPull1StepFL].lrZone4StartPos					:= ARDSUldZonePosOut[iPull1StepSFL].lrZone4StartPos - ARiVertArmPosOffset[iPull1StepFL];
						ARDs1StepUpDownMovement[iPull1StepFL].lrZone4EndPos					:= ARDSUldZonePosOut[iPull1StepSFL].lrZone4EndPos - ARiVertArmPosOffset[iPull1StepFL];
			
						ARDs1StepUpDownMovement[iPull1StepFL].lrMidPos							:= ARDSUldZonePosOut[iPull1StepSFL].lrMidPos;
			
						END_IF
					END_IF
				END_FOR
			END_IF


			(*No condition*)
			ARDs1StepUpDownMovement[iPull1StepFL].lrZone1SpeedVelo				:= fbA31ArmSpeedProfileMemory.ARDsArmSpeedProfileMemory[fbA21UpDownPattern.ARDsUpdownPatternMemory[ARi1StepPatternNo[iPull1StepFL]].iZone1SpdProfileNo].lrSpeedVelo;
			ARDs1StepUpDownMovement[iPull1StepFL].lrZone2SpeedVelo				:= fbA31ArmSpeedProfileMemory.ARDsArmSpeedProfileMemory[fbA21UpDownPattern.ARDsUpdownPatternMemory[ARi1StepPatternNo[iPull1StepFL]].iZone2SpdProfileNo].lrSpeedVelo;
			ARDs1StepUpDownMovement[iPull1StepFL].lrZone3SpeedVelo				:= fbA31ArmSpeedProfileMemory.ARDsArmSpeedProfileMemory[fbA21UpDownPattern.ARDsUpdownPatternMemory[ARi1StepPatternNo[iPull1StepFL]].iZone3SpdProfileNo].lrSpeedVelo;
			ARDs1StepUpDownMovement[iPull1StepFL].lrZone4SpeedVelo				:= fbA31ArmSpeedProfileMemory.ARDsArmSpeedProfileMemory[fbA21UpDownPattern.ARDsUpdownPatternMemory[ARi1StepPatternNo[iPull1StepFL]].iZone4SpdProfileNo].lrSpeedVelo;
			
			ARDs1StepUpDownMovement[iPull1StepFL].lrZone1Acc						:= fbA31ArmSpeedProfileMemory.ARDsArmSpeedProfileMemory[fbA21UpDownPattern.ARDsUpdownPatternMemory[ARi1StepPatternNo[iPull1StepFL]].iZone1SpdProfileNo].lrAcc;
			ARDs1StepUpDownMovement[iPull1StepFL].lrZone1Dcc						:= fbA31ArmSpeedProfileMemory.ARDsArmSpeedProfileMemory[fbA21UpDownPattern.ARDsUpdownPatternMemory[ARi1StepPatternNo[iPull1StepFL]].iZone1SpdProfileNo].lrDcc;
			ARDs1StepUpDownMovement[iPull1StepFL].lrZone2Acc						:= fbA31ArmSpeedProfileMemory.ARDsArmSpeedProfileMemory[fbA21UpDownPattern.ARDsUpdownPatternMemory[ARi1StepPatternNo[iPull1StepFL]].iZone2SpdProfileNo].lrAcc;
			ARDs1StepUpDownMovement[iPull1StepFL].lrZone2Dcc						:= fbA31ArmSpeedProfileMemory.ARDsArmSpeedProfileMemory[fbA21UpDownPattern.ARDsUpdownPatternMemory[ARi1StepPatternNo[iPull1StepFL]].iZone2SpdProfileNo].lrDcc;
			ARDs1StepUpDownMovement[iPull1StepFL].lrZone3Acc						:= fbA31ArmSpeedProfileMemory.ARDsArmSpeedProfileMemory[fbA21UpDownPattern.ARDsUpdownPatternMemory[ARi1StepPatternNo[iPull1StepFL]].iZone3SpdProfileNo].lrAcc;
			ARDs1StepUpDownMovement[iPull1StepFL].lrZone3Dcc						:= fbA31ArmSpeedProfileMemory.ARDsArmSpeedProfileMemory[fbA21UpDownPattern.ARDsUpdownPatternMemory[ARi1StepPatternNo[iPull1StepFL]].iZone3SpdProfileNo].lrDcc;
			ARDs1StepUpDownMovement[iPull1StepFL].lrZone4Acc						:= fbA31ArmSpeedProfileMemory.ARDsArmSpeedProfileMemory[fbA21UpDownPattern.ARDsUpdownPatternMemory[ARi1StepPatternNo[iPull1StepFL]].iZone4SpdProfileNo].lrAcc;
			ARDs1StepUpDownMovement[iPull1StepFL].lrZone4Dcc						:= fbA31ArmSpeedProfileMemory.ARDsArmSpeedProfileMemory[fbA21UpDownPattern.ARDsUpdownPatternMemory[ARi1StepPatternNo[iPull1StepFL]].iZone4SpdProfileNo].lrDcc;
			
			ARDs1StepUpDownMovement[iPull1StepFL].sReservedLreal;
			ARDs1StepUpDownMovement[iPull1StepFL].sUpDownPatternDescription	:= fbA21UpDownPattern.ARDsUpdownPatternMemory[ARi1StepPatternNo[iPull1StepFL]].sDescription;
	END_IF
END_FOR



(*[][][][][][][][][][][][][][][][][][][][][][][][][][][][][][][][][][][][][][][][][][][][][][][][][][][][][][][][][][][][][][][][][][][][][][][][][][][][][][][][][][][][][][][][][][][][][][][][][][][]*)
(*Call DS4StepUpDownMovement*)


(*1 Step UpDownMovement Data Pulling*)
iPull4StepFL := 1;

FOR iPull4StepFL := 1 TO iArmQty DO
	IF iPull4StepFL >=1 AND iPull4StepFL <= iArmQty THEN

			IF ARiCurrentHorzStnNo[iPull4StepFL] >= 1 AND ARiCurrentHorzStnNo[iPull4StepFL] <= iStnQty THEN
			ARDs4StepUpDownMovement[iPull4StepFL].lrZone1StartPos					:= ARDSStationZonePosOut[ARiCurrentHorzStnNo[iPull4StepFL]].lrZone1StartPos - ARiVertArmPosOffset[iPull4StepFL];
			ARDs4StepUpDownMovement[iPull4StepFL].lrZone1EndPos					:= ARDSStationZonePosOut[ARiCurrentHorzStnNo[iPull4StepFL]].lrZone1EndPos - ARiVertArmPosOffset[iPull4StepFL];
			ARDs4StepUpDownMovement[iPull4StepFL].lrZone2StartPos					:= ARDSStationZonePosOut[ARiCurrentHorzStnNo[iPull4StepFL]].lrZone2StartPos - ARiVertArmPosOffset[iPull4StepFL];
			ARDs4StepUpDownMovement[iPull4StepFL].lrZone2EndPos					:= ARDSStationZonePosOut[ARiCurrentHorzStnNo[iPull4StepFL]].lrZone2EndPos - ARiVertArmPosOffset[iPull4StepFL];
			ARDs4StepUpDownMovement[iPull4StepFL].lrZone3StartPos					:= ARDSStationZonePosOut[ARiCurrentHorzStnNo[iPull4StepFL]].lrZone3StartPos - ARiVertArmPosOffset[iPull4StepFL];
			ARDs4StepUpDownMovement[iPull4StepFL].lrZone3EndPos					:= ARDSStationZonePosOut[ARiCurrentHorzStnNo[iPull4StepFL]].lrZone3EndPos - ARiVertArmPosOffset[iPull4StepFL];
			ARDs4StepUpDownMovement[iPull4StepFL].lrZone4StartPos					:= ARDSStationZonePosOut[ARiCurrentHorzStnNo[iPull4StepFL]].lrZone4StartPos - ARiVertArmPosOffset[iPull4StepFL];
			ARDs4StepUpDownMovement[iPull4StepFL].lrZone4EndPos					:= ARDSStationZonePosOut[ARiCurrentHorzStnNo[iPull4StepFL]].lrZone4EndPos - ARiVertArmPosOffset[iPull4StepFL];
	
			ARDs4StepUpDownMovement[iPull4StepFL].lrMidPos							:= ARDSStationZonePosOut[ARiCurrentHorzStnNo[iPull4StepFL]].lrMidPos;
	
			ELSE

			iPull4StepSFL := 1;
				FOR iPull4StepSFL := 1 TO iLdStnQty DO
					IF iPull4StepSFL >=1 AND iPull4StepSFL <= iLdStnQty THEN

						(*With Condition*)
						IF ARiCurrentHorzStnNo[iPull4StepFL] = ARiLdStnID[iPull4StepSFL] THEN
						ARDs4StepUpDownMovement[iPull4StepFL].lrZone1StartPos					:= ARDSLdZonePosOut[iPull4StepSFL].lrZone1StartPos - ARiVertArmPosOffset[ARiCurrentHorzStnNo[iPull4StepFL]];
						ARDs4StepUpDownMovement[iPull4StepFL].lrZone1EndPos					:= ARDSLdZonePosOut[iPull4StepSFL].lrZone1EndPos - ARiVertArmPosOffset[ARiCurrentHorzStnNo[iPull4StepFL]];
						ARDs4StepUpDownMovement[iPull4StepFL].lrZone2StartPos					:= ARDSLdZonePosOut[iPull4StepSFL].lrZone2StartPos - ARiVertArmPosOffset[ARiCurrentHorzStnNo[iPull4StepFL]];
						ARDs4StepUpDownMovement[iPull4StepFL].lrZone2EndPos					:= ARDSLdZonePosOut[iPull4StepSFL].lrZone2EndPos - ARiVertArmPosOffset[ARiCurrentHorzStnNo[iPull4StepFL]];
						ARDs4StepUpDownMovement[iPull4StepFL].lrZone3StartPos					:= ARDSLdZonePosOut[iPull4StepSFL].lrZone3StartPos - ARiVertArmPosOffset[ARiCurrentHorzStnNo[iPull4StepFL]];
						ARDs4StepUpDownMovement[iPull4StepFL].lrZone3EndPos					:= ARDSLdZonePosOut[iPull4StepSFL].lrZone3EndPos - ARiVertArmPosOffset[ARiCurrentHorzStnNo[iPull4StepFL]];
						ARDs4StepUpDownMovement[iPull4StepFL].lrZone4StartPos					:= ARDSLdZonePosOut[iPull4StepSFL].lrZone4StartPos - ARiVertArmPosOffset[ARiCurrentHorzStnNo[iPull4StepFL]];
						ARDs4StepUpDownMovement[iPull4StepFL].lrZone4EndPos					:= ARDSLdZonePosOut[iPull4StepSFL].lrZone4EndPos - ARiVertArmPosOffset[ARiCurrentHorzStnNo[iPull4StepFL]];
			
						ARDs4StepUpDownMovement[iPull4StepFL].lrMidPos							:= ARDSLdZonePosOut[iPull4StepSFL].lrMidPos;
			
						END_IF
					END_IF
				END_FOR

			iPull4StepSFL := 1;
				FOR iPull4StepSFL := 1 TO iUldStnQty DO
					IF iPull4StepSFL >=1 AND iPull4StepSFL <= iUldStnQty THEN

						IF ARiCurrentHorzStnNo[iPull4StepFL] = ARiUldStnID[iPull4StepSFL] THEN
						ARDs4StepUpDownMovement[iPull4StepFL].lrZone1StartPos					:= ARDSUldZonePosOut[iPull4StepSFL].lrZone1StartPos - ARiVertArmPosOffset[iPull4StepFL];
						ARDs4StepUpDownMovement[iPull4StepFL].lrZone1EndPos					:= ARDSUldZonePosOut[iPull4StepSFL].lrZone1EndPos - ARiVertArmPosOffset[iPull4StepFL];
						ARDs4StepUpDownMovement[iPull4StepFL].lrZone2StartPos					:= ARDSUldZonePosOut[iPull4StepSFL].lrZone2StartPos - ARiVertArmPosOffset[iPull4StepFL];
						ARDs4StepUpDownMovement[iPull4StepFL].lrZone2EndPos					:= ARDSUldZonePosOut[iPull4StepSFL].lrZone2EndPos - ARiVertArmPosOffset[iPull4StepFL];
						ARDs4StepUpDownMovement[iPull4StepFL].lrZone3StartPos					:= ARDSUldZonePosOut[iPull4StepSFL].lrZone3StartPos - ARiVertArmPosOffset[iPull4StepFL];
						ARDs4StepUpDownMovement[iPull4StepFL].lrZone3EndPos					:= ARDSUldZonePosOut[iPull4StepSFL].lrZone3EndPos - ARiVertArmPosOffset[iPull4StepFL];
						ARDs4StepUpDownMovement[iPull4StepFL].lrZone4StartPos					:= ARDSUldZonePosOut[iPull4StepSFL].lrZone4StartPos - ARiVertArmPosOffset[iPull4StepFL];
						ARDs4StepUpDownMovement[iPull4StepFL].lrZone4EndPos					:= ARDSUldZonePosOut[iPull4StepSFL].lrZone4EndPos - ARiVertArmPosOffset[iPull4StepFL];
			
						ARDs4StepUpDownMovement[iPull4StepFL].lrMidPos							:= ARDSUldZonePosOut[iPull4StepSFL].lrMidPos;
			
						END_IF
					END_IF
				END_FOR

			END_IF
	

			(*No condition*)
			ARDs4StepUpDownMovement[iPull4StepFL].lrZone1SpeedVelo				:= fbA31ArmSpeedProfileMemory.ARDsArmSpeedProfileMemory[fbA21UpDownPattern.ARDsUpdownPatternMemory[ARi4StepPatternNo[iPull4StepFL]].iZone1SpdProfileNo].lrSpeedVelo;
			ARDs4StepUpDownMovement[iPull4StepFL].lrZone2SpeedVelo				:= fbA31ArmSpeedProfileMemory.ARDsArmSpeedProfileMemory[fbA21UpDownPattern.ARDsUpdownPatternMemory[ARi4StepPatternNo[iPull4StepFL]].iZone2SpdProfileNo].lrSpeedVelo;
			ARDs4StepUpDownMovement[iPull4StepFL].lrZone3SpeedVelo				:= fbA31ArmSpeedProfileMemory.ARDsArmSpeedProfileMemory[fbA21UpDownPattern.ARDsUpdownPatternMemory[ARi4StepPatternNo[iPull4StepFL]].iZone3SpdProfileNo].lrSpeedVelo;
			ARDs4StepUpDownMovement[iPull4StepFL].lrZone4SpeedVelo				:= fbA31ArmSpeedProfileMemory.ARDsArmSpeedProfileMemory[fbA21UpDownPattern.ARDsUpdownPatternMemory[ARi4StepPatternNo[iPull4StepFL]].iZone4SpdProfileNo].lrSpeedVelo;

